  STRUCT
   STAT0 : WORD ;
   STAT1 : WORD ;
   STAT2 : WORD ;
   STAT3 : WORD ;
   STAT4 : WORD ;
   STAT5 : WORD ;
   STAT6 : WORD ;
   STAT7 : WORD ;
   STAT8 : WORD ;
   STAT9 : WORD ;
   STAT10 : WORD ;
   STAT11 : WORD ;
   STAT12 : WORD ;
   STAT13 : WORD ;
   STAT14 : WORD ;
   STAT15 : WORD ;
   STAT16 : INT ;
   STAT17 : INT ;
   STAT18 : INT ;
   STAT19 : INT ;
   STAT20 : ARRAY  [1 .. 6 ] OF BYTE ;
   STAT21 : ARRAY  [1 .. 6 ] OF BYTE ;
   STAT22 : ARRAY  [1 .. 40 ] OF BOOL  := FALSE;
   STAT23 : ARRAY  [1 .. 40 ] OF BOOL  := FALSE;
   STAT24 : WORD ;
   STAT25 : WORD ;
   STAT26 : WORD ;
   STAT27 : WORD ;
   STAT28 : WORD ;
   STAT29 : WORD ;
   STAT30 : WORD ;
   STAT31 : ARRAY  [1 .. 7 ] OF WORD ;
   STAT32 : INT ;
   STAT33 : INT ;
   STAT34 : INT ;
   STAT35 : INT ;
   STAT36 : ARRAY  [1 .. 500 ] OF WORD ;
   STAT37 : ARRAY  [1 .. 16 ] OF BYTE ;
   STAT38 : ARRAY  [1 .. 4 ] OF BYTE ;
   STAT39 : ARRAY  [1 .. 16 ] OF BYTE ;
  END_STRUCT ;
BEGIN
   STAT0 := W#16#2714;
   STAT1 := W#16#87;
   STAT2 := W#16#2222;
   STAT3 := W#16#180;
   STAT4 := W#16#5416;
   STAT5 := W#16#60;
   STAT6 := W#16#0;
   STAT7 := W#16#0;
   STAT8 := W#16#87;
   STAT9 := W#16#2713;
   STAT10 := W#16#220A;
   STAT11 := W#16#8010;
   STAT12 := W#16#5254;
   STAT13 := W#16#4000;
   STAT14 := W#16#0;
   STAT15 := W#16#0;
   STAT16 := 0;
   STAT17 := 2;
   STAT18 := 3;
   STAT19 := 0;
   STAT20[1] := B#16#0;
   STAT20[2] := B#16#0;
   STAT20[3] := B#16#0;
   STAT20[4] := B#16#0;
   STAT20[5] := B#16#0;
   STAT20[6] := B#16#0;
   STAT21[1] := B#16#0;
   STAT21[2] := B#16#0;
   STAT21[3] := B#16#0;
   STAT21[4] := B#16#0;
   STAT21[5] := B#16#0;
   STAT21[6] := B#16#0;
   STAT22[1] := FALSE;
   STAT22[2] := FALSE;
   STAT22[3] := TRUE;
   STAT22[4] := FALSE;
   STAT22[5] := FALSE;
   STAT22[6] := FALSE;
   STAT22[7] := FALSE;
   STAT22[8] := TRUE;
   STAT22[9] := FALSE;
   STAT22[10] := FALSE;
   STAT22[11] := FALSE;
   STAT22[12] := FALSE;
   STAT22[13] := FALSE;
   STAT22[14] := FALSE;
   STAT22[15] := FALSE;
   STAT22[16] := FALSE;
   STAT22[17] := FALSE;
   STAT22[18] := FALSE;
   STAT22[19] := FALSE;
   STAT22[20] := FALSE;
   STAT22[21] := FALSE;
   STAT22[22] := FALSE;
   STAT22[23] := FALSE;
   STAT22[24] := FALSE;
   STAT22[25] := FALSE;
   STAT22[26] := FALSE;
   STAT22[27] := FALSE;
   STAT22[28] := FALSE;
   STAT22[29] := FALSE;
   STAT22[30] := FALSE;
   STAT22[31] := FALSE;
   STAT22[32] := FALSE;
   STAT22[33] := FALSE;
   STAT22[34] := FALSE;
   STAT22[35] := FALSE;
   STAT22[36] := FALSE;
   STAT22[37] := FALSE;
   STAT22[38] := FALSE;
   STAT22[39] := FALSE;
   STAT22[40] := FALSE;
   STAT23[1] := FALSE;
   STAT23[2] := TRUE;
   STAT23[3] := FALSE;
   STAT23[4] := FALSE;
   STAT23[5] := FALSE;
   STAT23[6] := TRUE;
   STAT23[7] := FALSE;
   STAT23[8] := FALSE;
   STAT23[9] := FALSE;
   STAT23[10] := FALSE;
   STAT23[11] := FALSE;
   STAT23[12] := FALSE;
   STAT23[13] := FALSE;
   STAT23[14] := FALSE;
   STAT23[15] := FALSE;
   STAT23[16] := FALSE;
   STAT23[17] := FALSE;
   STAT23[18] := FALSE;
   STAT23[19] := FALSE;
   STAT23[20] := FALSE;
   STAT23[21] := FALSE;
   STAT23[22] := FALSE;
   STAT23[23] := FALSE;
   STAT23[24] := FALSE;
   STAT23[25] := FALSE;
   STAT23[26] := FALSE;
   STAT23[27] := FALSE;
   STAT23[28] := FALSE;
   STAT23[29] := FALSE;
   STAT23[30] := FALSE;
   STAT23[31] := FALSE;
   STAT23[32] := FALSE;
   STAT23[33] := FALSE;
   STAT23[34] := FALSE;
   STAT23[35] := FALSE;
   STAT23[36] := FALSE;
   STAT23[37] := FALSE;
   STAT23[38] := FALSE;
   STAT23[39] := FALSE;
   STAT23[40] := FALSE;
   STAT24 := W#16#400;
   STAT25 := W#16#400;
   STAT26 := W#16#0;
   STAT27 := W#16#0;
   STAT28 := W#16#0;
   STAT29 := W#16#0;
   STAT30 := W#16#0;
   STAT31[1] := W#16#0;
   STAT31[2] := W#16#0;
   STAT31[3] := W#16#0;
   STAT31[4] := W#16#0;
   STAT31[5] := W#16#0;
   STAT31[6] := W#16#0;
   STAT31[7] := W#16#0;
   STAT32 := 100;
   STAT33 := 90;
   STAT34 := 80;
   STAT35 := 0;
   STAT36[1] := W#16#300;
   STAT36[2] := W#16#1418;
   STAT36[3] := W#16#3223;
   STAT36[4] := W#16#B;
   STAT36[5] := W#16#2713;
   STAT36[6] := W#16#200;
   STAT36[7] := W#16#1418;
   STAT36[8] := W#16#3221;
   STAT36[9] := W#16#1;
   STAT36[10] := W#16#2712;
   STAT36[11] := W#16#500;
   STAT36[12] := W#16#1418;
   STAT36[13] := W#16#3221;
   STAT36[14] := W#16#0;
   STAT36[15] := W#16#0;
   STAT36[16] := W#16#400;
   STAT36[17] := W#16#1418;
   STAT36[18] := W#16#3218;
   STAT36[19] := W#16#0;
   STAT36[20] := W#16#0;
   STAT36[21] := W#16#300;
   STAT36[22] := W#16#1418;
   STAT36[23] := W#16#2328;
   STAT36[24] := W#16#B;
   STAT36[25] := W#16#2712;
   STAT36[26] := W#16#200;
   STAT36[27] := W#16#1418;
   STAT36[28] := W#16#2327;
   STAT36[29] := W#16#1;
   STAT36[30] := W#16#2711;
   STAT36[31] := W#16#500;
   STAT36[32] := W#16#1418;
   STAT36[33] := W#16#2327;
   STAT36[34] := W#16#0;
   STAT36[35] := W#16#0;
   STAT36[36] := W#16#400;
   STAT36[37] := W#16#1418;
   STAT36[38] := W#16#2324;
   STAT36[39] := W#16#0;
   STAT36[40] := W#16#0;
   STAT36[41] := W#16#300;
   STAT36[42] := W#16#1418;
   STAT36[43] := W#16#2218;
   STAT36[44] := W#16#B;
   STAT36[45] := W#16#2711;
   STAT36[46] := W#16#200;
   STAT36[47] := W#16#1418;
   STAT36[48] := W#16#2217;
   STAT36[49] := W#16#1;
   STAT36[50] := W#16#2710;
   STAT36[51] := W#16#500;
   STAT36[52] := W#16#1418;
   STAT36[53] := W#16#2217;
   STAT36[54] := W#16#0;
   STAT36[55] := W#16#0;
   STAT36[56] := W#16#400;
   STAT36[57] := W#16#1418;
   STAT36[58] := W#16#2213;
   STAT36[59] := W#16#0;
   STAT36[60] := W#16#0;
   STAT36[61] := W#16#300;
   STAT36[62] := W#16#1418;
   STAT36[63] := W#16#2102;
   STAT36[64] := W#16#B;
   STAT36[65] := W#16#2710;
   STAT36[66] := W#16#200;
   STAT36[67] := W#16#1418;
   STAT36[68] := W#16#2101;
   STAT36[69] := W#16#1;
   STAT36[70] := W#16#2709;
   STAT36[71] := W#16#500;
   STAT36[72] := W#16#1418;
   STAT36[73] := W#16#2101;
   STAT36[74] := W#16#0;
   STAT36[75] := W#16#0;
   STAT36[76] := W#16#400;
   STAT36[77] := W#16#1418;
   STAT36[78] := W#16#2058;
   STAT36[79] := W#16#0;
   STAT36[80] := W#16#0;
   STAT36[81] := W#16#300;
   STAT36[82] := W#16#1418;
   STAT36[83] := W#16#1949;
   STAT36[84] := W#16#B;
   STAT36[85] := W#16#2709;
   STAT36[86] := W#16#200;
   STAT36[87] := W#16#1418;
   STAT36[88] := W#16#1948;
   STAT36[89] := W#16#1;
   STAT36[90] := W#16#2708;
   STAT36[91] := W#16#500;
   STAT36[92] := W#16#1418;
   STAT36[93] := W#16#1947;
   STAT36[94] := W#16#0;
   STAT36[95] := W#16#0;
   STAT36[96] := W#16#400;
   STAT36[97] := W#16#1418;
   STAT36[98] := W#16#1944;
   STAT36[99] := W#16#0;
   STAT36[100] := W#16#0;
   STAT36[101] := W#16#300;
   STAT36[102] := W#16#1418;
   STAT36[103] := W#16#1838;
   STAT36[104] := W#16#B;
   STAT36[105] := W#16#2708;
   STAT36[106] := W#16#200;
   STAT36[107] := W#16#1418;
   STAT36[108] := W#16#1837;
   STAT36[109] := W#16#1;
   STAT36[110] := W#16#2707;
   STAT36[111] := W#16#500;
   STAT36[112] := W#16#1418;
   STAT36[113] := W#16#1836;
   STAT36[114] := W#16#0;
   STAT36[115] := W#16#0;
   STAT36[116] := W#16#400;
   STAT36[117] := W#16#1418;
   STAT36[118] := W#16#1833;
   STAT36[119] := W#16#0;
   STAT36[120] := W#16#0;
   STAT36[121] := W#16#300;
   STAT36[122] := W#16#1418;
   STAT36[123] := W#16#1723;
   STAT36[124] := W#16#B;
   STAT36[125] := W#16#2707;
   STAT36[126] := W#16#200;
   STAT36[127] := W#16#1418;
   STAT36[128] := W#16#1721;
   STAT36[129] := W#16#1;
   STAT36[130] := W#16#2706;
   STAT36[131] := W#16#500;
   STAT36[132] := W#16#1418;
   STAT36[133] := W#16#1721;
   STAT36[134] := W#16#0;
   STAT36[135] := W#16#0;
   STAT36[136] := W#16#400;
   STAT36[137] := W#16#1418;
   STAT36[138] := W#16#1718;
   STAT36[139] := W#16#0;
   STAT36[140] := W#16#0;
   STAT36[141] := W#16#300;
   STAT36[142] := W#16#1418;
   STAT36[143] := W#16#1610;
   STAT36[144] := W#16#B;
   STAT36[145] := W#16#2706;
   STAT36[146] := W#16#200;
   STAT36[147] := W#16#1418;
   STAT36[148] := W#16#1609;
   STAT36[149] := W#16#1;
   STAT36[150] := W#16#2705;
   STAT36[151] := W#16#500;
   STAT36[152] := W#16#1418;
   STAT36[153] := W#16#1608;
   STAT36[154] := W#16#0;
   STAT36[155] := W#16#0;
   STAT36[156] := W#16#400;
   STAT36[157] := W#16#1418;
   STAT36[158] := W#16#1605;
   STAT36[159] := W#16#0;
   STAT36[160] := W#16#0;
   STAT36[161] := W#16#300;
   STAT36[162] := W#16#1418;
   STAT36[163] := W#16#1459;
   STAT36[164] := W#16#B;
   STAT36[165] := W#16#2705;
   STAT36[166] := W#16#200;
   STAT36[167] := W#16#1418;
   STAT36[168] := W#16#1458;
   STAT36[169] := W#16#1;
   STAT36[170] := W#16#2704;
   STAT36[171] := W#16#500;
   STAT36[172] := W#16#1418;
   STAT36[173] := W#16#1457;
   STAT36[174] := W#16#0;
   STAT36[175] := W#16#0;
   STAT36[176] := W#16#400;
   STAT36[177] := W#16#1418;
   STAT36[178] := W#16#1454;
   STAT36[179] := W#16#0;
   STAT36[180] := W#16#0;
   STAT36[181] := W#16#300;
   STAT36[182] := W#16#1418;
   STAT36[183] := W#16#1343;
   STAT36[184] := W#16#B;
   STAT36[185] := W#16#2704;
   STAT36[186] := W#16#200;
   STAT36[187] := W#16#1418;
   STAT36[188] := W#16#1342;
   STAT36[189] := W#16#1;
   STAT36[190] := W#16#2703;
   STAT36[191] := W#16#500;
   STAT36[192] := W#16#1418;
   STAT36[193] := W#16#1342;
   STAT36[194] := W#16#0;
   STAT36[195] := W#16#0;
   STAT36[196] := W#16#400;
   STAT36[197] := W#16#1418;
   STAT36[198] := W#16#1338;
   STAT36[199] := W#16#0;
   STAT36[200] := W#16#0;
   STAT36[201] := W#16#300;
   STAT36[202] := W#16#1418;
   STAT36[203] := W#16#1228;
   STAT36[204] := W#16#B;
   STAT36[205] := W#16#2703;
   STAT36[206] := W#16#200;
   STAT36[207] := W#16#1418;
   STAT36[208] := W#16#1226;
   STAT36[209] := W#16#1;
   STAT36[210] := W#16#2702;
   STAT36[211] := W#16#500;
   STAT36[212] := W#16#1418;
   STAT36[213] := W#16#1226;
   STAT36[214] := W#16#0;
   STAT36[215] := W#16#0;
   STAT36[216] := W#16#400;
   STAT36[217] := W#16#1418;
   STAT36[218] := W#16#1223;
   STAT36[219] := W#16#0;
   STAT36[220] := W#16#0;
   STAT36[221] := W#16#300;
   STAT36[222] := W#16#1418;
   STAT36[223] := W#16#1112;
   STAT36[224] := W#16#B;
   STAT36[225] := W#16#2702;
   STAT36[226] := W#16#200;
   STAT36[227] := W#16#1418;
   STAT36[228] := W#16#1111;
   STAT36[229] := W#16#1;
   STAT36[230] := W#16#2701;
   STAT36[231] := W#16#500;
   STAT36[232] := W#16#1418;
   STAT36[233] := W#16#1110;
   STAT36[234] := W#16#0;
   STAT36[235] := W#16#0;
   STAT36[236] := W#16#400;
   STAT36[237] := W#16#1418;
   STAT36[238] := W#16#1107;
   STAT36[239] := W#16#0;
   STAT36[240] := W#16#0;
   STAT36[241] := W#16#300;
   STAT36[242] := W#16#1418;
   STAT36[243] := W#16#957;
   STAT36[244] := W#16#B;
   STAT36[245] := W#16#2701;
   STAT36[246] := W#16#200;
   STAT36[247] := W#16#1418;
   STAT36[248] := W#16#955;
   STAT36[249] := W#16#1;
   STAT36[250] := W#16#2700;
   STAT36[251] := W#16#500;
   STAT36[252] := W#16#1418;
   STAT36[253] := W#16#955;
   STAT36[254] := W#16#0;
   STAT36[255] := W#16#0;
   STAT36[256] := W#16#400;
   STAT36[257] := W#16#1418;
   STAT36[258] := W#16#952;
   STAT36[259] := W#16#0;
   STAT36[260] := W#16#0;
   STAT36[261] := W#16#300;
   STAT36[262] := W#16#1418;
   STAT36[263] := W#16#844;
   STAT36[264] := W#16#B;
   STAT36[265] := W#16#2700;
   STAT36[266] := W#16#200;
   STAT36[267] := W#16#1418;
   STAT36[268] := W#16#843;
   STAT36[269] := W#16#1;
   STAT36[270] := W#16#2699;
   STAT36[271] := W#16#500;
   STAT36[272] := W#16#1418;
   STAT36[273] := W#16#842;
   STAT36[274] := W#16#0;
   STAT36[275] := W#16#0;
   STAT36[276] := W#16#400;
   STAT36[277] := W#16#1418;
   STAT36[278] := W#16#839;
   STAT36[279] := W#16#0;
   STAT36[280] := W#16#0;
   STAT36[281] := W#16#300;
   STAT36[282] := W#16#1418;
   STAT36[283] := W#16#729;
   STAT36[284] := W#16#B;
   STAT36[285] := W#16#2699;
   STAT36[286] := W#16#200;
   STAT36[287] := W#16#1418;
   STAT36[288] := W#16#728;
   STAT36[289] := W#16#1;
   STAT36[290] := W#16#2698;
   STAT36[291] := W#16#500;
   STAT36[292] := W#16#1418;
   STAT36[293] := W#16#728;
   STAT36[294] := W#16#0;
   STAT36[295] := W#16#0;
   STAT36[296] := W#16#400;
   STAT36[297] := W#16#1418;
   STAT36[298] := W#16#724;
   STAT36[299] := W#16#0;
   STAT36[300] := W#16#0;
   STAT36[301] := W#16#300;
   STAT36[302] := W#16#1418;
   STAT36[303] := W#16#324;
   STAT36[304] := W#16#B;
   STAT36[305] := W#16#2698;
   STAT36[306] := W#16#200;
   STAT36[307] := W#16#1418;
   STAT36[308] := W#16#322;
   STAT36[309] := W#16#1;
   STAT36[310] := W#16#2697;
   STAT36[311] := W#16#500;
   STAT36[312] := W#16#1418;
   STAT36[313] := W#16#322;
   STAT36[314] := W#16#0;
   STAT36[315] := W#16#0;
   STAT36[316] := W#16#400;
   STAT36[317] := W#16#1418;
   STAT36[318] := W#16#319;
   STAT36[319] := W#16#0;
   STAT36[320] := W#16#0;
   STAT36[321] := W#16#300;
   STAT36[322] := W#16#1418;
   STAT36[323] := W#16#211;
   STAT36[324] := W#16#B;
   STAT36[325] := W#16#2697;
   STAT36[326] := W#16#200;
   STAT36[327] := W#16#1418;
   STAT36[328] := W#16#209;
   STAT36[329] := W#16#1;
   STAT36[330] := W#16#2696;
   STAT36[331] := W#16#500;
   STAT36[332] := W#16#1418;
   STAT36[333] := W#16#209;
   STAT36[334] := W#16#0;
   STAT36[335] := W#16#0;
   STAT36[336] := W#16#400;
   STAT36[337] := W#16#1418;
   STAT36[338] := W#16#206;
   STAT36[339] := W#16#0;
   STAT36[340] := W#16#0;
   STAT36[341] := W#16#300;
   STAT36[342] := W#16#1418;
   STAT36[343] := W#16#55;
   STAT36[344] := W#16#B;
   STAT36[345] := W#16#2696;
   STAT36[346] := W#16#200;
   STAT36[347] := W#16#1418;
   STAT36[348] := W#16#53;
   STAT36[349] := W#16#1;
   STAT36[350] := W#16#2695;
   STAT36[351] := W#16#500;
   STAT36[352] := W#16#1418;
   STAT36[353] := W#16#53;
   STAT36[354] := W#16#0;
   STAT36[355] := W#16#0;
   STAT36[356] := W#16#400;
   STAT36[357] := W#16#1418;
   STAT36[358] := W#16#50;
   STAT36[359] := W#16#0;
   STAT36[360] := W#16#0;
   STAT36[361] := W#16#300;
   STAT36[362] := W#16#1417;
   STAT36[363] := W#16#5939;
   STAT36[364] := W#16#B;
   STAT36[365] := W#16#2695;
   STAT36[366] := W#16#200;
   STAT36[367] := W#16#1417;
   STAT36[368] := W#16#5938;
   STAT36[369] := W#16#1;
   STAT36[370] := W#16#2694;
   STAT36[371] := W#16#500;
   STAT36[372] := W#16#1417;
   STAT36[373] := W#16#5937;
   STAT36[374] := W#16#0;
   STAT36[375] := W#16#0;
   STAT36[376] := W#16#400;
   STAT36[377] := W#16#1417;
   STAT36[378] := W#16#5934;
   STAT36[379] := W#16#0;
   STAT36[380] := W#16#0;
   STAT36[381] := W#16#300;
   STAT36[382] := W#16#1417;
   STAT36[383] := W#16#5828;
   STAT36[384] := W#16#B;
   STAT36[385] := W#16#2694;
   STAT36[386] := W#16#200;
   STAT36[387] := W#16#1417;
   STAT36[388] := W#16#5827;
   STAT36[389] := W#16#1;
   STAT36[390] := W#16#2693;
   STAT36[391] := W#16#500;
   STAT36[392] := W#16#1417;
   STAT36[393] := W#16#5827;
   STAT36[394] := W#16#0;
   STAT36[395] := W#16#0;
   STAT36[396] := W#16#400;
   STAT36[397] := W#16#1417;
   STAT36[398] := W#16#5824;
   STAT36[399] := W#16#0;
   STAT36[400] := W#16#0;
   STAT36[401] := W#16#300;
   STAT36[402] := W#16#1417;
   STAT36[403] := W#16#5715;
   STAT36[404] := W#16#B;
   STAT36[405] := W#16#2693;
   STAT36[406] := W#16#200;
   STAT36[407] := W#16#1417;
   STAT36[408] := W#16#5714;
   STAT36[409] := W#16#1;
   STAT36[410] := W#16#2692;
   STAT36[411] := W#16#500;
   STAT36[412] := W#16#1417;
   STAT36[413] := W#16#5713;
   STAT36[414] := W#16#0;
   STAT36[415] := W#16#0;
   STAT36[416] := W#16#400;
   STAT36[417] := W#16#1417;
   STAT36[418] := W#16#5710;
   STAT36[419] := W#16#0;
   STAT36[420] := W#16#0;
   STAT36[421] := W#16#300;
   STAT36[422] := W#16#1417;
   STAT36[423] := W#16#5602;
   STAT36[424] := W#16#B;
   STAT36[425] := W#16#2692;
   STAT36[426] := W#16#200;
   STAT36[427] := W#16#1417;
   STAT36[428] := W#16#5601;
   STAT36[429] := W#16#1;
   STAT36[430] := W#16#2691;
   STAT36[431] := W#16#500;
   STAT36[432] := W#16#1417;
   STAT36[433] := W#16#5600;
   STAT36[434] := W#16#0;
   STAT36[435] := W#16#0;
   STAT36[436] := W#16#400;
   STAT36[437] := W#16#1417;
   STAT36[438] := W#16#5557;
   STAT36[439] := W#16#0;
   STAT36[440] := W#16#0;
   STAT36[441] := W#16#300;
   STAT36[442] := W#16#1417;
   STAT36[443] := W#16#5448;
   STAT36[444] := W#16#B;
   STAT36[445] := W#16#2691;
   STAT36[446] := W#16#200;
   STAT36[447] := W#16#1417;
   STAT36[448] := W#16#5447;
   STAT36[449] := W#16#1;
   STAT36[450] := W#16#2690;
   STAT36[451] := W#16#500;
   STAT36[452] := W#16#1417;
   STAT36[453] := W#16#5447;
   STAT36[454] := W#16#0;
   STAT36[455] := W#16#0;
   STAT36[456] := W#16#400;
   STAT36[457] := W#16#1417;
   STAT36[458] := W#16#5444;
   STAT36[459] := W#16#0;
   STAT36[460] := W#16#0;
   STAT36[461] := W#16#300;
   STAT36[462] := W#16#1417;
   STAT36[463] := W#16#5333;
   STAT36[464] := W#16#B;
   STAT36[465] := W#16#2690;
   STAT36[466] := W#16#200;
   STAT36[467] := W#16#1417;
   STAT36[468] := W#16#5331;
   STAT36[469] := W#16#1;
   STAT36[470] := W#16#2689;
   STAT36[471] := W#16#500;
   STAT36[472] := W#16#1417;
   STAT36[473] := W#16#5331;
   STAT36[474] := W#16#0;
   STAT36[475] := W#16#0;
   STAT36[476] := W#16#400;
   STAT36[477] := W#16#1417;
   STAT36[478] := W#16#5328;
   STAT36[479] := W#16#0;
   STAT36[480] := W#16#0;
   STAT36[481] := W#16#300;
   STAT36[482] := W#16#1417;
   STAT36[483] := W#16#5217;
   STAT36[484] := W#16#B;
   STAT36[485] := W#16#2689;
   STAT36[486] := W#16#200;
   STAT36[487] := W#16#1417;
   STAT36[488] := W#16#5216;
   STAT36[489] := W#16#1;
   STAT36[490] := W#16#2688;
   STAT36[491] := W#16#500;
   STAT36[492] := W#16#1417;
   STAT36[493] := W#16#5215;
   STAT36[494] := W#16#0;
   STAT36[495] := W#16#0;
   STAT36[496] := W#16#400;
   STAT36[497] := W#16#1417;
   STAT36[498] := W#16#5212;
   STAT36[499] := W#16#0;
   STAT36[500] := W#16#0;
   STAT37[1] := B#16#0;
   STAT37[2] := B#16#87;
   STAT37[3] := B#16#27;
   STAT37[4] := B#16#13;
   STAT37[5] := B#16#22;
   STAT37[6] := B#16#A;
   STAT37[7] := B#16#80;
   STAT37[8] := B#16#10;
   STAT37[9] := B#16#52;
   STAT37[10] := B#16#54;
   STAT37[11] := B#16#40;
   STAT37[12] := B#16#0;
   STAT37[13] := B#16#0;
   STAT37[14] := B#16#0;
   STAT37[15] := B#16#0;
   STAT37[16] := B#16#0;
   STAT38[1] := B#16#0;
   STAT38[2] := B#16#0;
   STAT38[3] := B#16#0;
   STAT38[4] := B#16#0;
   STAT39[1] := B#16#27;
   STAT39[2] := B#16#13;
   STAT39[3] := B#16#0;
   STAT39[4] := B#16#87;
   STAT39[5] := B#16#A;
   STAT39[6] := B#16#22;
   STAT39[7] := B#16#10;
   STAT39[8] := B#16#80;
   STAT39[9] := B#16#54;
   STAT39[10] := B#16#52;
   STAT39[11] := B#16#0;
   STAT39[12] := B#16#40;
   STAT39[13] := B#16#0;
   STAT39[14] := B#16#0;
   STAT39[15] := B#16#0;
   STAT39[16] := B#16#0;
END_DATA_BLOCK

DATA_BLOCK DB 169
VERSION : 0.1


  STRUCT
   STAT0 : WORD ;
   STAT1 : WORD ;
   STAT2 : WORD ;
   STAT3 : WORD ;
   STAT4 : WORD ;
   STAT5 : WORD ;
   STAT6 : WORD ;
   STAT7 : WORD ;
   STAT8 : WORD ;
   STAT9 : WORD ;
   STAT10 : WORD ;
   STAT11 : WORD ;
   STAT12 : WORD ;
   STAT13 : WORD ;
   STAT14 : WORD ;
   STAT15 : WORD ;
   STAT16 : INT ;
   STAT17 : INT ;
   STAT18 : INT ;
   STAT19 : INT ;
   STAT20 : ARRAY  [1 .. 6 ] OF BYTE ;
   STAT21 : ARRAY  [1 .. 6 ] OF BYTE ;
   STAT22 : ARRAY  [1 .. 40 ] OF BOOL  := FALSE;
   STAT23 : ARRAY  [1 .. 40 ] OF BOOL  := FALSE;
   STAT24 : WORD ;
   STAT25 : WORD ;
   STAT26 : WORD ;
   STAT27 : WORD ;
   STAT28 : WORD ;
   STAT29 : WORD ;
   STAT30 : WORD ;
   STAT31 : ARRAY  [1 .. 7 ] OF WORD ;
   STAT32 : INT ;
   STAT33 : INT ;
   STAT34 : INT ;
   STAT35 : INT ;
   STAT36 : ARRAY  [1 .. 500 ] OF WORD ;
   STAT37 : ARRAY  [1 .. 16 ] OF BYTE ;
   STAT38 : ARRAY  [1 .. 4 ] OF BYTE ;
   STAT39 : ARRAY  [1 .. 16 ] OF BYTE ;
  END_STRUCT ;
BEGIN
   STAT0 := W#16#2705;
   STAT1 := W#16#87;
   STAT2 := W#16#A22;
   STAT3 := W#16#1080;
   STAT4 := W#16#1026;
   STAT5 := W#16#40;
   STAT6 := W#16#0;
   STAT7 := W#16#0;
   STAT8 := W#16#87;
   STAT9 := W#16#2709;
   STAT10 := W#16#220A;
   STAT11 := W#16#8010;
   STAT12 := W#16#1610;
   STAT13 := W#16#4000;
   STAT14 := W#16#0;
   STAT15 := W#16#0;
   STAT16 := 2;
   STAT17 := 8;
   STAT18 := 3;
   STAT19 := 0;
   STAT20[1] := B#16#0;
   STAT20[2] := B#16#0;
   STAT20[3] := B#16#0;
   STAT20[4] := B#16#0;
   STAT20[5] := B#16#0;
   STAT20[6] := B#16#0;
   STAT21[1] := B#16#0;
   STAT21[2] := B#16#0;
   STAT21[3] := B#16#0;
   STAT21[4] := B#16#0;
   STAT21[5] := B#16#0;
   STAT21[6] := B#16#0;
   STAT22[1] := FALSE;
   STAT22[2] := FALSE;
   STAT22[3] := TRUE;
   STAT22[4] := FALSE;
   STAT22[5] := FALSE;
   STAT22[6] := FALSE;
   STAT22[7] := FALSE;
   STAT22[8] := TRUE;
   STAT22[9] := FALSE;
   STAT22[10] := FALSE;
   STAT22[11] := FALSE;
   STAT22[12] := FALSE;
   STAT22[13] := FALSE;
   STAT22[14] := FALSE;
   STAT22[15] := FALSE;
   STAT22[16] := FALSE;
   STAT22[17] := FALSE;
   STAT22[18] := FALSE;
   STAT22[19] := FALSE;
   STAT22[20] := FALSE;
   STAT22[21] := FALSE;
   STAT22[22] := FALSE;
   STAT22[23] := FALSE;
   STAT22[24] := FALSE;
   STAT22[25] := FALSE;
   STAT22[26] := FALSE;
   STAT22[27] := FALSE;
   STAT22[28] := FALSE;
   STAT22[29] := FALSE;
   STAT22[30] := FALSE;
   STAT22[31] := FALSE;
   STAT22[32] := FALSE;
   STAT22[33] := FALSE;
   STAT22[34] := FALSE;
   STAT22[35] := FALSE;
   STAT22[36] := FALSE;
   STAT22[37] := FALSE;
   STAT22[38] := FALSE;
   STAT22[39] := FALSE;
   STAT22[40] := FALSE;
   STAT23[1] := TRUE;
   STAT23[2] := FALSE;
   STAT23[3] := TRUE;
   STAT23[4] := TRUE;
   STAT23[5] := TRUE;
   STAT23[6] := FALSE;
   STAT23[7] := FALSE;
   STAT23[8] := FALSE;
   STAT23[9] := FALSE;
   STAT23[10] := FALSE;
   STAT23[11] := FALSE;
   STAT23[12] := FALSE;
   STAT23[13] := FALSE;
   STAT23[14] := FALSE;
   STAT23[15] := FALSE;
   STAT23[16] := FALSE;
   STAT23[17] := FALSE;
   STAT23[18] := FALSE;
   STAT23[19] := FALSE;
   STAT23[20] := FALSE;
   STAT23[21] := FALSE;
   STAT23[22] := FALSE;
   STAT23[23] := FALSE;
   STAT23[24] := FALSE;
   STAT23[25] := FALSE;
   STAT23[26] := TRUE;
   STAT23[27] := FALSE;
   STAT23[28] := FALSE;
   STAT23[29] := FALSE;
   STAT23[30] := FALSE;
   STAT23[31] := FALSE;
   STAT23[32] := FALSE;
   STAT23[33] := FALSE;
   STAT23[34] := FALSE;
   STAT23[35] := FALSE;
   STAT23[36] := FALSE;
   STAT23[37] := FALSE;
   STAT23[38] := FALSE;
   STAT23[39] := FALSE;
   STAT23[40] := FALSE;
   STAT24 := W#16#0;
   STAT25 := W#16#0;
   STAT26 := W#16#0;
   STAT27 := W#16#0;
   STAT28 := W#16#0;
   STAT29 := W#16#0;
   STAT30 := W#16#0;
   STAT31[1] := W#16#0;
   STAT31[2] := W#16#0;
   STAT31[3] := W#16#0;
   STAT31[4] := W#16#0;
   STAT31[5] := W#16#0;
   STAT31[6] := W#16#0;
   STAT31[7] := W#16#0;
   STAT32 := 100;
   STAT33 := 90;
   STAT34 := 80;
   STAT35 := 0;
   STAT36[1] := W#16#400;
   STAT36[2] := W#16#1418;
   STAT36[3] := W#16#3243;
   STAT36[4] := W#16#0;
   STAT36[5] := W#16#2709;
   STAT36[6] := W#16#300;
   STAT36[7] := W#16#1418;
   STAT36[8] := W#16#3240;
   STAT36[9] := W#16#B;
   STAT36[10] := W#16#2705;
   STAT36[11] := W#16#200;
   STAT36[12] := W#16#1418;
   STAT36[13] := W#16#3238;
   STAT36[14] := W#16#1;
   STAT36[15] := W#16#0;
   STAT36[16] := W#16#500;
   STAT36[17] := W#16#1418;
   STAT36[18] := W#16#3229;
   STAT36[19] := W#16#0;
   STAT36[20] := W#16#0;
   STAT36[21] := W#16#400;
   STAT36[22] := W#16#1418;
   STAT36[23] := W#16#3229;
   STAT36[24] := W#16#0;
   STAT36[25] := W#16#0;
   STAT36[26] := W#16#500;
   STAT36[27] := W#16#1418;
   STAT36[28] := W#16#3228;
   STAT36[29] := W#16#0;
   STAT36[30] := W#16#0;
   STAT36[31] := W#16#400;
   STAT36[32] := W#16#1418;
   STAT36[33] := W#16#3128;
   STAT36[34] := W#16#0;
   STAT36[35] := W#16#2708;
   STAT36[36] := W#16#300;
   STAT36[37] := W#16#1418;
   STAT36[38] := W#16#3125;
   STAT36[39] := W#16#B;
   STAT36[40] := W#16#2704;
   STAT36[41] := W#16#200;
   STAT36[42] := W#16#1418;
   STAT36[43] := W#16#3124;
   STAT36[44] := W#16#1;
   STAT36[45] := W#16#0;
   STAT36[46] := W#16#500;
   STAT36[47] := W#16#1418;
   STAT36[48] := W#16#3115;
   STAT36[49] := W#16#0;
   STAT36[50] := W#16#0;
   STAT36[51] := W#16#400;
   STAT36[52] := W#16#1418;
   STAT36[53] := W#16#3114;
   STAT36[54] := W#16#0;
   STAT36[55] := W#16#0;
   STAT36[56] := W#16#500;
   STAT36[57] := W#16#1418;
   STAT36[58] := W#16#3113;
   STAT36[59] := W#16#0;
   STAT36[60] := W#16#0;
   STAT36[61] := W#16#400;
   STAT36[62] := W#16#1418;
   STAT36[63] := W#16#2233;
   STAT36[64] := W#16#0;
   STAT36[65] := W#16#2707;
   STAT36[66] := W#16#300;
   STAT36[67] := W#16#1418;
   STAT36[68] := W#16#2231;
   STAT36[69] := W#16#B;
   STAT36[70] := W#16#2703;
   STAT36[71] := W#16#200;
   STAT36[72] := W#16#1418;
   STAT36[73] := W#16#2229;
   STAT36[74] := W#16#1;
   STAT36[75] := W#16#0;
   STAT36[76] := W#16#500;
   STAT36[77] := W#16#1418;
   STAT36[78] := W#16#2217;
   STAT36[79] := W#16#0;
   STAT36[80] := W#16#0;
   STAT36[81] := W#16#400;
   STAT36[82] := W#16#1418;
   STAT36[83] := W#16#2216;
   STAT36[84] := W#16#0;
   STAT36[85] := W#16#0;
   STAT36[86] := W#16#500;
   STAT36[87] := W#16#1418;
   STAT36[88] := W#16#2215;
   STAT36[89] := W#16#0;
   STAT36[90] := W#16#0;
   STAT36[91] := W#16#400;
   STAT36[92] := W#16#1418;
   STAT36[93] := W#16#2123;
   STAT36[94] := W#16#0;
   STAT36[95] := W#16#2706;
   STAT36[96] := W#16#300;
   STAT36[97] := W#16#1418;
   STAT36[98] := W#16#2120;
   STAT36[99] := W#16#B;
   STAT36[100] := W#16#2702;
   STAT36[101] := W#16#200;
   STAT36[102] := W#16#1418;
   STAT36[103] := W#16#2119;
   STAT36[104] := W#16#1;
   STAT36[105] := W#16#0;
   STAT36[106] := W#16#500;
   STAT36[107] := W#16#1418;
   STAT36[108] := W#16#2103;
   STAT36[109] := W#16#0;
   STAT36[110] := W#16#0;
   STAT36[111] := W#16#400;
   STAT36[112] := W#16#1418;
   STAT36[113] := W#16#2007;
   STAT36[114] := W#16#0;
   STAT36[115] := W#16#2705;
   STAT36[116] := W#16#300;
   STAT36[117] := W#16#1418;
   STAT36[118] := W#16#2004;
   STAT36[119] := W#16#B;
   STAT36[120] := W#16#2701;
   STAT36[121] := W#16#200;
   STAT36[122] := W#16#1418;
   STAT36[123] := W#16#2003;
   STAT36[124] := W#16#1;
   STAT36[125] := W#16#0;
   STAT36[126] := W#16#500;
   STAT36[127] := W#16#1418;
   STAT36[128] := W#16#1949;
   STAT36[129] := W#16#0;
   STAT36[130] := W#16#0;
   STAT36[131] := W#16#400;
   STAT36[132] := W#16#1418;
   STAT36[133] := W#16#1948;
   STAT36[134] := W#16#0;
   STAT36[135] := W#16#0;
   STAT36[136] := W#16#500;
   STAT36[137] := W#16#1418;
   STAT36[138] := W#16#1947;
   STAT36[139] := W#16#0;
   STAT36[140] := W#16#0;
   STAT36[141] := W#16#400;
   STAT36[142] := W#16#1418;
   STAT36[143] := W#16#1854;
   STAT36[144] := W#16#0;
   STAT36[145] := W#16#2704;
   STAT36[146] := W#16#300;
   STAT36[147] := W#16#1418;
   STAT36[148] := W#16#1851;
   STAT36[149] := W#16#B;
   STAT36[150] := W#16#2700;
   STAT36[151] := W#16#200;
   STAT36[152] := W#16#1418;
   STAT36[153] := W#16#1849;
   STAT36[154] := W#16#1;
   STAT36[155] := W#16#0;
   STAT36[156] := W#16#500;
   STAT36[157] := W#16#1418;
   STAT36[158] := W#16#1833;
   STAT36[159] := W#16#0;
   STAT36[160] := W#16#0;
   STAT36[161] := W#16#400;
   STAT36[162] := W#16#1418;
   STAT36[163] := W#16#1833;
   STAT36[164] := W#16#0;
   STAT36[165] := W#16#0;
   STAT36[166] := W#16#500;
   STAT36[167] := W#16#1418;
   STAT36[168] := W#16#1832;
   STAT36[169] := W#16#0;
   STAT36[170] := W#16#0;
   STAT36[171] := W#16#400;
   STAT36[172] := W#16#1418;
   STAT36[173] := W#16#1743;
   STAT36[174] := W#16#0;
   STAT36[175] := W#16#2703;
   STAT36[176] := W#16#300;
   STAT36[177] := W#16#1418;
   STAT36[178] := W#16#1740;
   STAT36[179] := W#16#B;
   STAT36[180] := W#16#2699;
   STAT36[181] := W#16#200;
   STAT36[182] := W#16#1418;
   STAT36[183] := W#16#1739;
   STAT36[184] := W#16#1;
   STAT36[185] := W#16#0;
   STAT36[186] := W#16#500;
   STAT36[187] := W#16#1418;
   STAT36[188] := W#16#1721;
   STAT36[189] := W#16#0;
   STAT36[190] := W#16#0;
   STAT36[191] := W#16#400;
   STAT36[192] := W#16#1418;
   STAT36[193] := W#16#1720;
   STAT36[194] := W#16#0;
   STAT36[195] := W#16#0;
   STAT36[196] := W#16#500;
   STAT36[197] := W#16#1418;
   STAT36[198] := W#16#1719;
   STAT36[199] := W#16#0;
   STAT36[200] := W#16#0;
   STAT36[201] := W#16#400;
   STAT36[202] := W#16#1418;
   STAT36[203] := W#16#1627;
   STAT36[204] := W#16#0;
   STAT36[205] := W#16#2702;
   STAT36[206] := W#16#300;
   STAT36[207] := W#16#1418;
   STAT36[208] := W#16#1625;
   STAT36[209] := W#16#B;
   STAT36[210] := W#16#2698;
   STAT36[211] := W#16#200;
   STAT36[212] := W#16#1418;
   STAT36[213] := W#16#1623;
   STAT36[214] := W#16#1;
   STAT36[215] := W#16#0;
   STAT36[216] := W#16#500;
   STAT36[217] := W#16#1418;
   STAT36[218] := W#16#1607;
   STAT36[219] := W#16#0;
   STAT36[220] := W#16#0;
   STAT36[221] := W#16#400;
   STAT36[222] := W#16#1418;
   STAT36[223] := W#16#1607;
   STAT36[224] := W#16#0;
   STAT36[225] := W#16#0;
   STAT36[226] := W#16#500;
   STAT36[227] := W#16#1418;
   STAT36[228] := W#16#1606;
   STAT36[229] := W#16#0;
   STAT36[230] := W#16#0;
   STAT36[231] := W#16#400;
   STAT36[232] := W#16#1418;
   STAT36[233] := W#16#1514;
   STAT36[234] := W#16#0;
   STAT36[235] := W#16#2701;
   STAT36[236] := W#16#300;
   STAT36[237] := W#16#1418;
   STAT36[238] := W#16#1511;
   STAT36[239] := W#16#B;
   STAT36[240] := W#16#2697;
   STAT36[241] := W#16#200;
   STAT36[242] := W#16#1418;
   STAT36[243] := W#16#1510;
   STAT36[244] := W#16#1;
   STAT36[245] := W#16#0;
   STAT36[246] := W#16#500;
   STAT36[247] := W#16#1418;
   STAT36[248] := W#16#1454;
   STAT36[249] := W#16#0;
   STAT36[250] := W#16#0;
   STAT36[251] := W#16#400;
   STAT36[252] := W#16#1418;
   STAT36[253] := W#16#1454;
   STAT36[254] := W#16#0;
   STAT36[255] := W#16#0;
   STAT36[256] := W#16#500;
   STAT36[257] := W#16#1418;
   STAT36[258] := W#16#1453;
   STAT36[259] := W#16#0;
   STAT36[260] := W#16#0;
   STAT36[261] := W#16#400;
   STAT36[262] := W#16#1418;
   STAT36[263] := W#16#1404;
   STAT36[264] := W#16#0;
   STAT36[265] := W#16#2700;
   STAT36[266] := W#16#300;
   STAT36[267] := W#16#1418;
   STAT36[268] := W#16#1401;
   STAT36[269] := W#16#B;
   STAT36[270] := W#16#2696;
   STAT36[271] := W#16#200;
   STAT36[272] := W#16#1418;
   STAT36[273] := W#16#1359;
   STAT36[274] := W#16#1;
   STAT36[275] := W#16#0;
   STAT36[276] := W#16#500;
   STAT36[277] := W#16#1418;
   STAT36[278] := W#16#1342;
   STAT36[279] := W#16#0;
   STAT36[280] := W#16#0;
   STAT36[281] := W#16#400;
   STAT36[282] := W#16#1418;
   STAT36[283] := W#16#1342;
   STAT36[284] := W#16#0;
   STAT36[285] := W#16#0;
   STAT36[286] := W#16#500;
   STAT36[287] := W#16#1418;
   STAT36[288] := W#16#1340;
   STAT36[289] := W#16#0;
   STAT36[290] := W#16#0;
   STAT36[291] := W#16#400;
   STAT36[292] := W#16#1418;
   STAT36[293] := W#16#1248;
   STAT36[294] := W#16#0;
   STAT36[295] := W#16#2699;
   STAT36[296] := W#16#300;
   STAT36[297] := W#16#1418;
   STAT36[298] := W#16#1245;
   STAT36[299] := W#16#B;
   STAT36[300] := W#16#2695;
   STAT36[301] := W#16#200;
   STAT36[302] := W#16#1418;
   STAT36[303] := W#16#1244;
   STAT36[304] := W#16#1;
   STAT36[305] := W#16#0;
   STAT36[306] := W#16#500;
   STAT36[307] := W#16#1418;
   STAT36[308] := W#16#1228;
   STAT36[309] := W#16#0;
   STAT36[310] := W#16#0;
   STAT36[311] := W#16#400;
   STAT36[312] := W#16#1418;
   STAT36[313] := W#16#1227;
   STAT36[314] := W#16#0;
   STAT36[315] := W#16#0;
   STAT36[316] := W#16#500;
   STAT36[317] := W#16#1418;
   STAT36[318] := W#16#1226;
   STAT36[319] := W#16#0;
   STAT36[320] := W#16#0;
   STAT36[321] := W#16#400;
   STAT36[322] := W#16#1418;
   STAT36[323] := W#16#1132;
   STAT36[324] := W#16#0;
   STAT36[325] := W#16#2698;
   STAT36[326] := W#16#300;
   STAT36[327] := W#16#1418;
   STAT36[328] := W#16#1130;
   STAT36[329] := W#16#B;
   STAT36[330] := W#16#2694;
   STAT36[331] := W#16#200;
   STAT36[332] := W#16#1418;
   STAT36[333] := W#16#1128;
   STAT36[334] := W#16#1;
   STAT36[335] := W#16#0;
   STAT36[336] := W#16#500;
   STAT36[337] := W#16#1418;
   STAT36[338] := W#16#1115;
   STAT36[339] := W#16#0;
   STAT36[340] := W#16#0;
   STAT36[341] := W#16#400;
   STAT36[342] := W#16#1418;
   STAT36[343] := W#16#1114;
   STAT36[344] := W#16#0;
   STAT36[345] := W#16#0;
   STAT36[346] := W#16#500;
   STAT36[347] := W#16#1418;
   STAT36[348] := W#16#1113;
   STAT36[349] := W#16#0;
   STAT36[350] := W#16#0;
   STAT36[351] := W#16#400;
   STAT36[352] := W#16#1418;
   STAT36[353] := W#16#1016;
   STAT36[354] := W#16#0;
   STAT36[355] := W#16#2697;
   STAT36[356] := W#16#300;
   STAT36[357] := W#16#1418;
   STAT36[358] := W#16#1014;
   STAT36[359] := W#16#B;
   STAT36[360] := W#16#2693;
   STAT36[361] := W#16#200;
   STAT36[362] := W#16#1418;
   STAT36[363] := W#16#1012;
   STAT36[364] := W#16#1;
   STAT36[365] := W#16#0;
   STAT36[366] := W#16#500;
   STAT36[367] := W#16#1418;
   STAT36[368] := W#16#1002;
   STAT36[369] := W#16#0;
   STAT36[370] := W#16#0;
   STAT36[371] := W#16#400;
   STAT36[372] := W#16#1418;
   STAT36[373] := W#16#901;
   STAT36[374] := W#16#0;
   STAT36[375] := W#16#2696;
   STAT36[376] := W#16#300;
   STAT36[377] := W#16#1418;
   STAT36[378] := W#16#858;
   STAT36[379] := W#16#B;
   STAT36[380] := W#16#2692;
   STAT36[381] := W#16#200;
   STAT36[382] := W#16#1418;
   STAT36[383] := W#16#857;
   STAT36[384] := W#16#1;
   STAT36[385] := W#16#0;
   STAT36[386] := W#16#500;
   STAT36[387] := W#16#1418;
   STAT36[388] := W#16#848;
   STAT36[389] := W#16#0;
   STAT36[390] := W#16#0;
   STAT36[391] := W#16#400;
   STAT36[392] := W#16#1418;
   STAT36[393] := W#16#848;
   STAT36[394] := W#16#0;
   STAT36[395] := W#16#0;
   STAT36[396] := W#16#500;
   STAT36[397] := W#16#1418;
   STAT36[398] := W#16#846;
   STAT36[399] := W#16#0;
   STAT36[400] := W#16#0;
   STAT36[401] := W#16#400;
   STAT36[402] := W#16#1418;
   STAT36[403] := W#16#749;
   STAT36[404] := W#16#0;
   STAT36[405] := W#16#2695;
   STAT36[406] := W#16#300;
   STAT36[407] := W#16#1418;
   STAT36[408] := W#16#746;
   STAT36[409] := W#16#B;
   STAT36[410] := W#16#2691;
   STAT36[411] := W#16#200;
   STAT36[412] := W#16#1418;
   STAT36[413] := W#16#744;
   STAT36[414] := W#16#1;
   STAT36[415] := W#16#0;
   STAT36[416] := W#16#500;
   STAT36[417] := W#16#1418;
   STAT36[418] := W#16#735;
   STAT36[419] := W#16#0;
   STAT36[420] := W#16#0;
   STAT36[421] := W#16#400;
   STAT36[422] := W#16#1418;
   STAT36[423] := W#16#735;
   STAT36[424] := W#16#0;
   STAT36[425] := W#16#0;
   STAT36[426] := W#16#500;
   STAT36[427] := W#16#1418;
   STAT36[428] := W#16#734;
   STAT36[429] := W#16#0;
   STAT36[430] := W#16#0;
   STAT36[431] := W#16#400;
   STAT36[432] := W#16#1418;
   STAT36[433] := W#16#634;
   STAT36[434] := W#16#0;
   STAT36[435] := W#16#2694;
   STAT36[436] := W#16#300;
   STAT36[437] := W#16#1418;
   STAT36[438] := W#16#632;
   STAT36[439] := W#16#B;
   STAT36[440] := W#16#2690;
   STAT36[441] := W#16#200;
   STAT36[442] := W#16#1418;
   STAT36[443] := W#16#630;
   STAT36[444] := W#16#1;
   STAT36[445] := W#16#0;
   STAT36[446] := W#16#500;
   STAT36[447] := W#16#1418;
   STAT36[448] := W#16#621;
   STAT36[449] := W#16#0;
   STAT36[450] := W#16#0;
   STAT36[451] := W#16#400;
   STAT36[452] := W#16#1418;
   STAT36[453] := W#16#620;
   STAT36[454] := W#16#0;
   STAT36[455] := W#16#0;
   STAT36[456] := W#16#500;
   STAT36[457] := W#16#1418;
   STAT36[458] := W#16#619;
   STAT36[459] := W#16#0;
   STAT36[460] := W#16#0;
   STAT36[461] := W#16#400;
   STAT36[462] := W#16#1418;
   STAT36[463] := W#16#228;
   STAT36[464] := W#16#0;
   STAT36[465] := W#16#2693;
   STAT36[466] := W#16#300;
   STAT36[467] := W#16#1418;
   STAT36[468] := W#16#226;
   STAT36[469] := W#16#B;
   STAT36[470] := W#16#2689;
   STAT36[471] := W#16#200;
   STAT36[472] := W#16#1418;
   STAT36[473] := W#16#224;
   STAT36[474] := W#16#1;
   STAT36[475] := W#16#0;
   STAT36[476] := W#16#500;
   STAT36[477] := W#16#1418;
   STAT36[478] := W#16#215;
   STAT36[479] := W#16#0;
   STAT36[480] := W#16#0;
   STAT36[481] := W#16#400;
   STAT36[482] := W#16#1418;
   STAT36[483] := W#16#215;
   STAT36[484] := W#16#0;
   STAT36[485] := W#16#0;
   STAT36[486] := W#16#500;
   STAT36[487] := W#16#1418;
   STAT36[488] := W#16#213;
   STAT36[489] := W#16#0;
   STAT36[490] := W#16#0;
   STAT36[491] := W#16#400;
   STAT36[492] := W#16#1418;
   STAT36[493] := W#16#115;
   STAT36[494] := W#16#0;
   STAT36[495] := W#16#2692;
   STAT36[496] := W#16#300;
   STAT36[497] := W#16#1418;
   STAT36[498] := W#16#112;
   STAT36[499] := W#16#B;
   STAT36[500] := W#16#2688;
   STAT37[1] := B#16#0;
   STAT37[2] := B#16#87;
   STAT37[3] := B#16#27;
   STAT37[4] := B#16#5;
   STAT37[5] := B#16#22;
   STAT37[6] := B#16#A;
   STAT37[7] := B#16#80;
   STAT37[8] := B#16#10;
   STAT37[9] := B#16#26;
   STAT37[10] := B#16#10;
   STAT37[11] := B#16#40;
   STAT37[12] := B#16#0;
   STAT37[13] := B#16#0;
   STAT37[14] := B#16#0;
   STAT37[15] := B#16#0;
   STAT37[16] := B#16#0;
   STAT38[1] := B#16#0;
   STAT38[2] := B#16#0;
   STAT38[3] := B#16#0;
   STAT38[4] := B#16#0;
   STAT39[1] := B#16#27;
   STAT39[2] := B#16#9;
   STAT39[3] := B#16#0;
   STAT39[4] := B#16#87;
   STAT39[5] := B#16#A;
   STAT39[6] := B#16#22;
   STAT39[7] := B#16#10;
   STAT39[8] := B#16#80;
   STAT39[9] := B#16#10;
   STAT39[10] := B#16#16;
   STAT39[11] := B#16#0;
   STAT39[12] := B#16#40;
   STAT39[13] := B#16#0;
   STAT39[14] := B#16#0;
   STAT39[15] := B#16#0;
   STAT39[16] := B#16#0;
END_DATA_BLOCK

DATA_BLOCK DB 170
VERSION : 0.1


  STRUCT
   STAT0 : WORD ;
   STAT1 : WORD ;
   STAT2 : WORD ;
   STAT3 : WORD ;
   STAT4 : WORD ;
   STAT5 : WORD ;
   STAT6 : WORD ;
   STAT7 : WORD ;
   STAT8 : WORD ;
   STAT9 : WORD ;
   STAT10 : WORD ;
   STAT11 : WORD ;
   STAT12 : WORD ;
   STAT13 : WORD ;
   STAT14 : WORD ;
   STAT15 : WORD ;
   STAT16 : INT ;
   STAT17 : INT ;
   STAT18 : INT ;
   STAT19 : INT ;
   STAT20 : ARRAY  [1 .. 6 ] OF BYTE ;
   STAT21 : ARRAY  [1 .. 6 ] OF BYTE ;
   STAT22 : ARRAY  [1 .. 40 ] OF BOOL  := FALSE;
   STAT23 : ARRAY  [1 .. 40 ] OF BOOL  := FALSE;
   STAT24 : WORD ;
   STAT25 : WORD ;
   STAT26 : WORD ;
   STAT27 : WORD ;
   STAT28 : WORD ;
   STAT29 : WORD ;
   STAT30 : WORD ;
   STAT31 : ARRAY  [1 .. 7 ] OF WORD ;
   STAT32 : INT ;
   STAT33 : INT ;
   STAT34 : INT ;
   STAT35 : INT ;
   STAT36 : ARRAY  [1 .. 500 ] OF WORD ;
   STAT37 : ARRAY  [1 .. 16 ] OF BYTE ;
   STAT38 : ARRAY  [1 .. 4 ] OF BYTE ;
   STAT39 : ARRAY  [1 .. 16 ] OF BYTE ;
  END_STRUCT ;
BEGIN
   STAT0 := W#16#0;
   STAT1 := W#16#0;
   STAT2 := W#16#0;
   STAT3 := W#16#0;
   STAT4 := W#16#0;
   STAT5 := W#16#0;
   STAT6 := W#16#0;
   STAT7 := W#16#0;
   STAT8 := W#16#0;
   STAT9 := W#16#0;
   STAT10 := W#16#0;
   STAT11 := W#16#0;
   STAT12 := W#16#0;
   STAT13 := W#16#0;
   STAT14 := W#16#0;
   STAT15 := W#16#0;
   STAT16 := 0;
   STAT17 := 0;
   STAT18 := 0;
   STAT19 := 0;
   STAT20[1] := B#16#0;
   STAT20[2] := B#16#0;
   STAT20[3] := B#16#0;
   STAT20[4] := B#16#0;
   STAT20[5] := B#16#0;
   STAT20[6] := B#16#0;
   STAT21[1] := B#16#0;
   STAT21[2] := B#16#0;
   STAT21[3] := B#16#0;
   STAT21[4] := B#16#0;
   STAT21[5] := B#16#0;
   STAT21[6] := B#16#0;
   STAT22[1] := FALSE;
   STAT22[2] := FALSE;
   STAT22[3] := FALSE;
   STAT22[4] := FALSE;
   STAT22[5] := FALSE;
   STAT22[6] := FALSE;
   STAT22[7] := FALSE;
   STAT22[8] := FALSE;
   STAT22[9] := FALSE;
   STAT22[10] := FALSE;
   STAT22[11] := FALSE;
   STAT22[12] := FALSE;
   STAT22[13] := FALSE;
   STAT22[14] := FALSE;
   STAT22[15] := FALSE;
   STAT22[16] := FALSE;
   STAT22[17] := FALSE;
   STAT22[18] := FALSE;
   STAT22[19] := FALSE;
   STAT22[20] := FALSE;
   STAT22[21] := FALSE;
   STAT22[22] := FALSE;
   STAT22[23] := FALSE;
   STAT22[24] := FALSE;
   STAT22[25] := FALSE;
   STAT22[26] := FALSE;
   STAT22[27] := FALSE;
   STAT22[28] := FALSE;
   STAT22[29] := FALSE;
   STAT22[30] := FALSE;
   STAT22[31] := FALSE;
   STAT22[32] := FALSE;
   STAT22[33] := FALSE;
   STAT22[34] := FALSE;
   STAT22[35] := FALSE;
   STAT22[36] := FALSE;
   STAT22[37] := FALSE;
   STAT22[38] := FALSE;
   STAT22[39] := FALSE;
   STAT22[40] := FALSE;
   STAT23[1] := FALSE;
   STAT23[2] := FALSE;
   STAT23[3] := FALSE;
   STAT23[4] := FALSE;
   STAT23[5] := FALSE;
   STAT23[6] := FALSE;
   STAT23[7] := FALSE;
   STAT23[8] := FALSE;
   STAT23[9] := FALSE;
   STAT23[10] := FALSE;
   STAT23[11] := FALSE;
   STAT23[12] := FALSE;
   STAT23[13] := FALSE;
   STAT23[14] := FALSE;
   STAT23[15] := FALSE;
   STAT23[16] := FALSE;
   STAT23[17] := FALSE;
   STAT23[18] := FALSE;
   STAT23[19] := FALSE;
   STAT23[20] := FALSE;
   STAT23[21] := FALSE;
   STAT23[22] := FALSE;
   STAT23[23] := FALSE;
   STAT23[24] := FALSE;
   STAT23[25] := FALSE;
   STAT23[26] := FALSE;
   STAT23[27] := FALSE;
   STAT23[28] := FALSE;
   STAT23[29] := FALSE;
   STAT23[30] := FALSE;
   STAT23[31] := FALSE;
   STAT23[32] := FALSE;
   STAT23[33] := FALSE;
   STAT23[34] := FALSE;
   STAT23[35] := FALSE;
   STAT23[36] := FALSE;
   STAT23[37] := FALSE;
   STAT23[38] := FALSE;
   STAT23[39] := FALSE;
   STAT23[40] := FALSE;
   STAT24 := W#16#0;
   STAT25 := W#16#0;
   STAT26 := W#16#0;
   STAT27 := W#16#0;
   STAT28 := W#16#0;
   STAT29 := W#16#0;
   STAT30 := W#16#0;
   STAT31[1] := W#16#0;
   STAT31[2] := W#16#0;
   STAT31[3] := W#16#0;
   STAT31[4] := W#16#0;
   STAT31[5] := W#16#0;
   STAT31[6] := W#16#0;
   STAT31[7] := W#16#0;
   STAT32 := 0;
   STAT33 := 0;
   STAT34 := 0;
   STAT35 := 0;
   STAT36[1] := W#16#0;
   STAT36[2] := W#16#0;
   STAT36[3] := W#16#0;
   STAT36[4] := W#16#0;
   STAT36[5] := W#16#0;
   STAT36[6] := W#16#0;
   STAT36[7] := W#16#0;
   STAT36[8] := W#16#0;
   STAT36[9] := W#16#0;
   STAT36[10] := W#16#0;
   STAT36[11] := W#16#0;
   STAT36[12] := W#16#0;
   STAT36[13] := W#16#0;
   STAT36[14] := W#16#0;
   STAT36[15] := W#16#0;
   STAT36[16] := W#16#0;
   STAT36[17] := W#16#0;
   STAT36[18] := W#16#0;
   STAT36[19] := W#16#0;
   STAT36[20] := W#16#0;
   STAT36[21] := W#16#0;
   STAT36[22] := W#16#0;
   STAT36[23] := W#16#0;
   STAT36[24] := W#16#0;
   STAT36[25] := W#16#0;
   STAT36[26] := W#16#0;
   STAT36[27] := W#16#0;
   STAT36[28] := W#16#0;
   STAT36[29] := W#16#0;
   STAT36[30] := W#16#0;
   STAT36[31] := W#16#0;
   STAT36[32] := W#16#0;
   STAT36[33] := W#16#0;
   STAT36[34] := W#16#0;
   STAT36[35] := W#16#0;
   STAT36[36] := W#16#0;
   STAT36[37] := W#16#0;
   STAT36[38] := W#16#0;
   STAT36[39] := W#16#0;
   STAT36[40] := W#16#0;
   STAT36[41] := W#16#0;
   STAT36[42] := W#16#0;
   STAT36[43] := W#16#0;
   STAT36[44] := W#16#0;
   STAT36[45] := W#16#0;
   STAT36[46] := W#16#0;
   STAT36[47] := W#16#0;
   STAT36[48] := W#16#0;
   STAT36[49] := W#16#0;
   STAT36[50] := W#16#0;
   STAT36[51] := W#16#0;
   STAT36[52] := W#16#0;
   STAT36[53] := W#16#0;
   STAT36[54] := W#16#0;
   STAT36[55] := W#16#0;
   STAT36[56] := W#16#0;
   STAT36[57] := W#16#0;
   STAT36[58] := W#16#0;
   STAT36[59] := W#16#0;
   STAT36[60] := W#16#0;
   STAT36[61] := W#16#0;
   STAT36[62] := W#16#0;
   STAT36[63] := W#16#0;
   STAT36[64] := W#16#0;
   STAT36[65] := W#16#0;
   STAT36[66] := W#16#0;
   STAT36[67] := W#16#0;
   STAT36[68] := W#16#0;
   STAT36[69] := W#16#0;
   STAT36[70] := W#16#0;
   STAT36[71] := W#16#0;
   STAT36[72] := W#16#0;
   STAT36[73] := W#16#0;
   STAT36[74] := W#16#0;
   STAT36[75] := W#16#0;
   STAT36[76] := W#16#0;
   STAT36[77] := W#16#0;
   STAT36[78] := W#16#0;
   STAT36[79] := W#16#0;
   STAT36[80] := W#16#0;
   STAT36[81] := W#16#0;
   STAT36[82] := W#16#0;
   STAT36[83] := W#16#0;
   STAT36[84] := W#16#0;
   STAT36[85] := W#16#0;
   STAT36[86] := W#16#0;
   STAT36[87] := W#16#0;
   STAT36[88] := W#16#0;
   STAT36[89] := W#16#0;
   STAT36[90] := W#16#0;
   STAT36[91] := W#16#0;
   STAT36[92] := W#16#0;
   STAT36[93] := W#16#0;
   STAT36[94] := W#16#0;
   STAT36[95] := W#16#0;
   STAT36[96] := W#16#0;
   STAT36[97] := W#16#0;
   STAT36[98] := W#16#0;
   STAT36[99] := W#16#0;
   STAT36[100] := W#16#0;
   STAT36[101] := W#16#0;
   STAT36[102] := W#16#0;
   STAT36[103] := W#16#0;
   STAT36[104] := W#16#0;
   STAT36[105] := W#16#0;
   STAT36[106] := W#16#0;
   STAT36[107] := W#16#0;
   STAT36[108] := W#16#0;
   STAT36[109] := W#16#0;
   STAT36[110] := W#16#0;
   STAT36[111] := W#16#0;
   STAT36[112] := W#16#0;
   STAT36[113] := W#16#0;
   STAT36[114] := W#16#0;
   STAT36[115] := W#16#0;
   STAT36[116] := W#16#0;
   STAT36[117] := W#16#0;
   STAT36[118] := W#16#0;
   STAT36[119] := W#16#0;
   STAT36[120] := W#16#0;
   STAT36[121] := W#16#0;
   STAT36[122] := W#16#0;
   STAT36[123] := W#16#0;
   STAT36[124] := W#16#0;
   STAT36[125] := W#16#0;
   STAT36[126] := W#16#0;
   STAT36[127] := W#16#0;
   STAT36[128] := W#16#0;
   STAT36[129] := W#16#0;
   STAT36[130] := W#16#0;
   STAT36[131] := W#16#0;
   STAT36[132] := W#16#0;
   STAT36[133] := W#16#0;
   STAT36[134] := W#16#0;
   STAT36[135] := W#16#0;
   STAT36[136] := W#16#0;
   STAT36[137] := W#16#0;
   STAT36[138] := W#16#0;
   STAT36[139] := W#16#0;
   STAT36[140] := W#16#0;
   STAT36[141] := W#16#0;
   STAT36[142] := W#16#0;
   STAT36[143] := W#16#0;
   STAT36[144] := W#16#0;
   STAT36[145] := W#16#0;
   STAT36[146] := W#16#0;
   STAT36[147] := W#16#0;
   STAT36[148] := W#16#0;
   STAT36[149] := W#16#0;
   STAT36[150] := W#16#0;
   STAT36[151] := W#16#0;
   STAT36[152] := W#16#0;
   STAT36[153] := W#16#0;
   STAT36[154] := W#16#0;
   STAT36[155] := W#16#0;
   STAT36[156] := W#16#0;
   STAT36[157] := W#16#0;
   STAT36[158] := W#16#0;
   STAT36[159] := W#16#0;
   STAT36[160] := W#16#0;
   STAT36[161] := W#16#0;
   STAT36[162] := W#16#0;
   STAT36[163] := W#16#0;
   STAT36[164] := W#16#0;
   STAT36[165] := W#16#0;
   STAT36[166] := W#16#0;
   STAT36[167] := W#16#0;
   STAT36[168] := W#16#0;
   STAT36[169] := W#16#0;
   STAT36[170] := W#16#0;
   STAT36[171] := W#16#0;
   STAT36[172] := W#16#0;
   STAT36[173] := W#16#0;
   STAT36[174] := W#16#0;
   STAT36[175] := W#16#0;
   STAT36[176] := W#16#0;
   STAT36[177] := W#16#0;
   STAT36[178] := W#16#0;
   STAT36[179] := W#16#0;
   STAT36[180] := W#16#0;
   STAT36[181] := W#16#0;
   STAT36[182] := W#16#0;
   STAT36[183] := W#16#0;
   STAT36[184] := W#16#0;
   STAT36[185] := W#16#0;
   STAT36[186] := W#16#0;
   STAT36[187] := W#16#0;
   STAT36[188] := W#16#0;
   STAT36[189] := W#16#0;
   STAT36[190] := W#16#0;
   STAT36[191] := W#16#0;
   STAT36[192] := W#16#0;
   STAT36[193] := W#16#0;
   STAT36[194] := W#16#0;
   STAT36[195] := W#16#0;
   STAT36[196] := W#16#0;
   STAT36[197] := W#16#0;
   STAT36[198] := W#16#0;
   STAT36[199] := W#16#0;
   STAT36[200] := W#16#0;
   STAT36[201] := W#16#0;
   STAT36[202] := W#16#0;
   STAT36[203] := W#16#0;
   STAT36[204] := W#16#0;
   STAT36[205] := W#16#0;
   STAT36[206] := W#16#0;
   STAT36[207] := W#16#0;
   STAT36[208] := W#16#0;
   STAT36[209] := W#16#0;
   STAT36[210] := W#16#0;
   STAT36[211] := W#16#0;
   STAT36[212] := W#16#0;
   STAT36[213] := W#16#0;
   STAT36[214] := W#16#0;
   STAT36[215] := W#16#0;
   STAT36[216] := W#16#0;
   STAT36[217] := W#16#0;
   STAT36[218] := W#16#0;
   STAT36[219] := W#16#0;
   STAT36[220] := W#16#0;
   STAT36[221] := W#16#0;
   STAT36[222] := W#16#0;
   STAT36[223] := W#16#0;
   STAT36[224] := W#16#0;
   STAT36[225] := W#16#0;
   STAT36[226] := W#16#0;
   STAT36[227] := W#16#0;
   STAT36[228] := W#16#0;
   STAT36[229] := W#16#0;
   STAT36[230] := W#16#0;
   STAT36[231] := W#16#0;
   STAT36[232] := W#16#0;
   STAT36[233] := W#16#0;
   STAT36[234] := W#16#0;
   STAT36[235] := W#16#0;
   STAT36[236] := W#16#0;
   STAT36[237] := W#16#0;
   STAT36[238] := W#16#0;
   STAT36[239] := W#16#0;
   STAT36[240] := W#16#0;
   STAT36[241] := W#16#0;
   STAT36[242] := W#16#0;
   STAT36[243] := W#16#0;
   STAT36[244] := W#16#0;
   STAT36[245] := W#16#0;
   STAT36[246] := W#16#0;
   STAT36[247] := W#16#0;
   STAT36[248] := W#16#0;
   STAT36[249] := W#16#0;
   STAT36[250] := W#16#0;
   STAT36[251] := W#16#0;
   STAT36[252] := W#16#0;
   STAT36[253] := W#16#0;
   STAT36[254] := W#16#0;
   STAT36[255] := W#16#0;
   STAT36[256] := W#16#0;
   STAT36[257] := W#16#0;
   STAT36[258] := W#16#0;
   STAT36[259] := W#16#0;
   STAT36[260] := W#16#0;
   STAT36[261] := W#16#0;
   STAT36[262] := W#16#0;
   STAT36[263] := W#16#0;
   STAT36[264] := W#16#0;
   STAT36[265] := W#16#0;
   STAT36[266] := W#16#0;
   STAT36[267] := W#16#0;
   STAT36[268] := W#16#0;
   STAT36[269] := W#16#0;
   STAT36[270] := W#16#0;
   STAT36[271] := W#16#0;
   STAT36[272] := W#16#0;
   STAT36[273] := W#16#0;
   STAT36[274] := W#16#0;
   STAT36[275] := W#16#0;
   STAT36[276] := W#16#0;
   STAT36[277] := W#16#0;
   STAT36[278] := W#16#0;
   STAT36[279] := W#16#0;
   STAT36[280] := W#16#0;
   STAT36[281] := W#16#0;
   STAT36[282] := W#16#0;
   STAT36[283] := W#16#0;
   STAT36[284] := W#16#0;
   STAT36[285] := W#16#0;
   STAT36[286] := W#16#0;
   STAT36[287] := W#16#0;
   STAT36[288] := W#16#0;
   STAT36[289] := W#16#0;
   STAT36[290] := W#16#0;
   STAT36[291] := W#16#0;
   STAT36[292] := W#16#0;
   STAT36[293] := W#16#0;
   STAT36[294] := W#16#0;
   STAT36[295] := W#16#0;
   STAT36[296] := W#16#0;
   STAT36[297] := W#16#0;
   STAT36[298] := W#16#0;
   STAT36[299] := W#16#0;
   STAT36[300] := W#16#0;
   STAT36[301] := W#16#0;
   STAT36[302] := W#16#0;
   STAT36[303] := W#16#0;
   STAT36[304] := W#16#0;
   STAT36[305] := W#16#0;
   STAT36[306] := W#16#0;
   STAT36[307] := W#16#0;
   STAT36[308] := W#16#0;
   STAT36[309] := W#16#0;
   STAT36[310] := W#16#0;
   STAT36[311] := W#16#0;
   STAT36[312] := W#16#0;
   STAT36[313] := W#16#0;
   STAT36[314] := W#16#0;
   STAT36[315] := W#16#0;
   STAT36[316] := W#16#0;
   STAT36[317] := W#16#0;
   STAT36[318] := W#16#0;
   STAT36[319] := W#16#0;
   STAT36[320] := W#16#0;
   STAT36[321] := W#16#0;
   STAT36[322] := W#16#0;
   STAT36[323] := W#16#0;
   STAT36[324] := W#16#0;
   STAT36[325] := W#16#0;
   STAT36[326] := W#16#0;
   STAT36[327] := W#16#0;
   STAT36[328] := W#16#0;
   STAT36[329] := W#16#0;
   STAT36[330] := W#16#0;
   STAT36[331] := W#16#0;
   STAT36[332] := W#16#0;
   STAT36[333] := W#16#0;
   STAT36[334] := W#16#0;
   STAT36[335] := W#16#0;
   STAT36[336] := W#16#0;
   STAT36[337] := W#16#0;
   STAT36[338] := W#16#0;
   STAT36[339] := W#16#0;
   STAT36[340] := W#16#0;
   STAT36[341] := W#16#0;
   STAT36[342] := W#16#0;
   STAT36[343] := W#16#0;
   STAT36[344] := W#16#0;
   STAT36[345] := W#16#0;
   STAT36[346] := W#16#0;
   STAT36[347] := W#16#0;
   STAT36[348] := W#16#0;
   STAT36[349] := W#16#0;
   STAT36[350] := W#16#0;
   STAT36[351] := W#16#0;
   STAT36[352] := W#16#0;
   STAT36[353] := W#16#0;
   STAT36[354] := W#16#0;
   STAT36[355] := W#16#0;
   STAT36[356] := W#16#0;
   STAT36[357] := W#16#0;
   STAT36[358] := W#16#0;
   STAT36[359] := W#16#0;
   STAT36[360] := W#16#0;
   STAT36[361] := W#16#0;
   STAT36[362] := W#16#0;
   STAT36[363] := W#16#0;
   STAT36[364] := W#16#0;
   STAT36[365] := W#16#0;
   STAT36[366] := W#16#0;
   STAT36[367] := W#16#0;
   STAT36[368] := W#16#0;
   STAT36[369] := W#16#0;
   STAT36[370] := W#16#0;
   STAT36[371] := W#16#0;
   STAT36[372] := W#16#0;
   STAT36[373] := W#16#0;
   STAT36[374] := W#16#0;
   STAT36[375] := W#16#0;
   STAT36[376] := W#16#0;
   STAT36[377] := W#16#0;
   STAT36[378] := W#16#0;
   STAT36[379] := W#16#0;
   STAT36[380] := W#16#0;
   STAT36[381] := W#16#0;
   STAT36[382] := W#16#0;
   STAT36[383] := W#16#0;
   STAT36[384] := W#16#0;
   STAT36[385] := W#16#0;
   STAT36[386] := W#16#0;
   STAT36[387] := W#16#0;
   STAT36[388] := W#16#0;
   STAT36[389] := W#16#0;
   STAT36[390] := W#16#0;
   STAT36[391] := W#16#0;
   STAT36[392] := W#16#0;
   STAT36[393] := W#16#0;
   STAT36[394] := W#16#0;
   STAT36[395] := W#16#0;
   STAT36[396] := W#16#0;
   STAT36[397] := W#16#0;
   STAT36[398] := W#16#0;
   STAT36[399] := W#16#0;
   STAT36[400] := W#16#0;
   STAT36[401] := W#16#0;
   STAT36[402] := W#16#0;
   STAT36[403] := W#16#0;
   STAT36[404] := W#16#0;
   STAT36[405] := W#16#0;
   STAT36[406] := W#16#0;
   STAT36[407] := W#16#0;
   STAT36[408] := W#16#0;
   STAT36[409] := W#16#0;
   STAT36[410] := W#16#0;
   STAT36[411] := W#16#0;
   STAT36[412] := W#16#0;
   STAT36[413] := W#16#0;
   STAT36[414] := W#16#0;
   STAT36[415] := W#16#0;
   STAT36[416] := W#16#0;
   STAT36[417] := W#16#0;
   STAT36[418] := W#16#0;
   STAT36[419] := W#16#0;
   STAT36[420] := W#16#0;
   STAT36[421] := W#16#0;
   STAT36[422] := W#16#0;
   STAT36[423] := W#16#0;
   STAT36[424] := W#16#0;
   STAT36[425] := W#16#0;
   STAT36[426] := W#16#0;
   STAT36[427] := W#16#0;
   STAT36[428] := W#16#0;
   STAT36[429] := W#16#0;
   STAT36[430] := W#16#0;
   STAT36[431] := W#16#0;
   STAT36[432] := W#16#0;
   STAT36[433] := W#16#0;
   STAT36[434] := W#16#0;
   STAT36[435] := W#16#0;
   STAT36[436] := W#16#0;
   STAT36[437] := W#16#0;
   STAT36[438] := W#16#0;
   STAT36[439] := W#16#0;
   STAT36[440] := W#16#0;
   STAT36[441] := W#16#0;
   STAT36[442] := W#16#0;
   STAT36[443] := W#16#0;
   STAT36[444] := W#16#0;
   STAT36[445] := W#16#0;
   STAT36[446] := W#16#0;
   STAT36[447] := W#16#0;
   STAT36[448] := W#16#0;
   STAT36[449] := W#16#0;
   STAT36[450] := W#16#0;
   STAT36[451] := W#16#0;
   STAT36[452] := W#16#0;
   STAT36[453] := W#16#0;
   STAT36[454] := W#16#0;
   STAT36[455] := W#16#0;
   STAT36[456] := W#16#0;
   STAT36[457] := W#16#0;
   STAT36[458] := W#16#0;
   STAT36[459] := W#16#0;
   STAT36[460] := W#16#0;
   STAT36[461] := W#16#0;
   STAT36[462] := W#16#0;
   STAT36[463] := W#16#0;
   STAT36[464] := W#16#0;
   STAT36[465] := W#16#0;
   STAT36[466] := W#16#0;
   STAT36[467] := W#16#0;
   STAT36[468] := W#16#0;
   STAT36[469] := W#16#0;
   STAT36[470] := W#16#0;
   STAT36[471] := W#16#0;
   STAT36[472] := W#16#0;
   STAT36[473] := W#16#0;
   STAT36[474] := W#16#0;
   STAT36[475] := W#16#0;
   STAT36[476] := W#16#0;
   STAT36[477] := W#16#0;
   STAT36[478] := W#16#0;
   STAT36[479] := W#16#0;
   STAT36[480] := W#16#0;
   STAT36[481] := W#16#0;
   STAT36[482] := W#16#0;
   STAT36[483] := W#16#0;
   STAT36[484] := W#16#0;
   STAT36[485] := W#16#0;
   STAT36[486] := W#16#0;
   STAT36[487] := W#16#0;
   STAT36[488] := W#16#0;
   STAT36[489] := W#16#0;
   STAT36[490] := W#16#0;
   STAT36[491] := W#16#0;
   STAT36[492] := W#16#0;
   STAT36[493] := W#16#0;
   STAT36[494] := W#16#0;
   STAT36[495] := W#16#0;
   STAT36[496] := W#16#0;
   STAT36[497] := W#16#0;
   STAT36[498] := W#16#0;
   STAT36[499] := W#16#0;
   STAT36[500] := W#16#0;
   STAT37[1] := B#16#0;
   STAT37[2] := B#16#0;
   STAT37[3] := B#16#0;
   STAT37[4] := B#16#0;
   STAT37[5] := B#16#0;
   STAT37[6] := B#16#0;
   STAT37[7] := B#16#0;
   STAT37[8] := B#16#0;
   STAT37[9] := B#16#0;
   STAT37[10] := B#16#0;
   STAT37[11] := B#16#0;
   STAT37[12] := B#16#0;
   STAT37[13] := B#16#0;
   STAT37[14] := B#16#0;
   STAT37[15] := B#16#0;
   STAT37[16] := B#16#0;
   STAT38[1] := B#16#0;
   STAT38[2] := B#16#0;
   STAT38[3] := B#16#0;
   STAT38[4] := B#16#0;
   STAT39[1] := B#16#0;
   STAT39[2] := B#16#0;
   STAT39[3] := B#16#0;
   STAT39[4] := B#16#0;
   STAT39[5] := B#16#0;
   STAT39[6] := B#16#0;
   STAT39[7] := B#16#0;
   STAT39[8] := B#16#0;
   STAT39[9] := B#16#0;
   STAT39[10] := B#16#0;
   STAT39[11] := B#16#0;
   STAT39[12] := B#16#0;
   STAT39[13] := B#16#0;
   STAT39[14] := B#16#0;
   STAT39[15] := B#16#0;
   STAT39[16] := B#16#0;
END_DATA_BLOCK

DATA_BLOCK DB 171
VERSION : 0.1


  STRUCT
   STAT0 : ARRAY  [1 .. 320 ] OF BYTE ;
   STAT1 : INT ;
   STAT2 : WORD ;
   STAT3 : INT ;
   STAT4 : INT ;
   STAT5 : INT ;
   STAT6 : INT ;
   STAT7 : INT ;
   STAT8 : INT ;
   STAT9 : INT ;
   STAT10 : INT ;
   STAT11 : INT ;
   STAT12 : INT ;
   STAT13 : INT ;
   STAT14 : INT ;
   STAT15 : INT ;
   STAT16 : INT ;
   STAT17 : INT ;
   STAT18 : INT ;
   STAT19 : INT ;
   STAT20 : INT ;
   STAT21 : ARRAY  [1 .. 20 ] OF WORD ;
  END_STRUCT ;
BEGIN
   STAT0[1] := B#16#0;
   STAT0[2] := B#16#87;
   STAT0[3] := B#16#27;
   STAT0[4] := B#16#16;
   STAT0[5] := B#16#22;
   STAT0[6] := B#16#22;
   STAT0[7] := B#16#80;
   STAT0[8] := B#16#4;
   STAT0[9] := B#16#16;
   STAT0[10] := B#16#10;
   STAT0[11] := B#16#60;
   STAT0[12] := B#16#0;
   STAT0[13] := B#16#0;
   STAT0[14] := B#16#0;
   STAT0[15] := B#16#0;
   STAT0[16] := B#16#0;
   STAT0[17] := B#16#0;
   STAT0[18] := B#16#87;
   STAT0[19] := B#16#27;
   STAT0[20] := B#16#15;
   STAT0[21] := B#16#22;
   STAT0[22] := B#16#22;
   STAT0[23] := B#16#80;
   STAT0[24] := B#16#1;
   STAT0[25] := B#16#62;
   STAT0[26] := B#16#54;
   STAT0[27] := B#16#60;
   STAT0[28] := B#16#0;
   STAT0[29] := B#16#0;
   STAT0[30] := B#16#0;
   STAT0[31] := B#16#0;
   STAT0[32] := B#16#0;
   STAT0[33] := B#16#0;
   STAT0[34] := B#16#87;
   STAT0[35] := B#16#27;
   STAT0[36] := B#16#14;
   STAT0[37] := B#16#22;
   STAT0[38] := B#16#22;
   STAT0[39] := B#16#80;
   STAT0[40] := B#16#1;
   STAT0[41] := B#16#16;
   STAT0[42] := B#16#54;
   STAT0[43] := B#16#60;
   STAT0[44] := B#16#0;
   STAT0[45] := B#16#0;
   STAT0[46] := B#16#0;
   STAT0[47] := B#16#0;
   STAT0[48] := B#16#0;
   STAT0[49] := B#16#0;
   STAT0[50] := B#16#87;
   STAT0[51] := B#16#27;
   STAT0[52] := B#16#13;
   STAT0[53] := B#16#22;
   STAT0[54] := B#16#A;
   STAT0[55] := B#16#80;
   STAT0[56] := B#16#10;
   STAT0[57] := B#16#52;
   STAT0[58] := B#16#54;
   STAT0[59] := B#16#40;
   STAT0[60] := B#16#0;
   STAT0[61] := B#16#0;
   STAT0[62] := B#16#0;
   STAT0[63] := B#16#0;
   STAT0[64] := B#16#0;
   STAT0[65] := B#16#0;
   STAT0[66] := B#16#87;
   STAT0[67] := B#16#27;
   STAT0[68] := B#16#12;
   STAT0[69] := B#16#22;
   STAT0[70] := B#16#22;
   STAT0[71] := B#16#80;
   STAT0[72] := B#16#1;
   STAT0[73] := B#16#26;
   STAT0[74] := B#16#54;
   STAT0[75] := B#16#60;
   STAT0[76] := B#16#0;
   STAT0[77] := B#16#0;
   STAT0[78] := B#16#0;
   STAT0[79] := B#16#0;
   STAT0[80] := B#16#0;
   STAT0[81] := B#16#0;
   STAT0[82] := B#16#87;
   STAT0[83] := B#16#27;
   STAT0[84] := B#16#11;
   STAT0[85] := B#16#22;
   STAT0[86] := B#16#84;
   STAT0[87] := B#16#80;
   STAT0[88] := B#16#1;
   STAT0[89] := B#16#62;
   STAT0[90] := B#16#54;
   STAT0[91] := B#16#40;
   STAT0[92] := B#16#0;
   STAT0[93] := B#16#0;
   STAT0[94] := B#16#0;
   STAT0[95] := B#16#0;
   STAT0[96] := B#16#0;
   STAT0[97] := B#16#0;
   STAT0[98] := B#16#87;
   STAT0[99] := B#16#27;
   STAT0[100] := B#16#10;
   STAT0[101] := B#16#22;
   STAT0[102] := B#16#22;
   STAT0[103] := B#16#80;
   STAT0[104] := B#16#1;
   STAT0[105] := B#16#52;
   STAT0[106] := B#16#54;
   STAT0[107] := B#16#60;
   STAT0[108] := B#16#0;
   STAT0[109] := B#16#0;
   STAT0[110] := B#16#0;
   STAT0[111] := B#16#0;
   STAT0[112] := B#16#0;
   STAT0[113] := B#16#0;
   STAT0[114] := B#16#87;
   STAT0[115] := B#16#27;
   STAT0[116] := B#16#9;
   STAT0[117] := B#16#22;
   STAT0[118] := B#16#A;
   STAT0[119] := B#16#80;
   STAT0[120] := B#16#10;
   STAT0[121] := B#16#16;
   STAT0[122] := B#16#10;
   STAT0[123] := B#16#40;
   STAT0[124] := B#16#0;
   STAT0[125] := B#16#0;
   STAT0[126] := B#16#0;
   STAT0[127] := B#16#0;
   STAT0[128] := B#16#0;
   STAT0[129] := B#16#0;
   STAT0[130] := B#16#0;
   STAT0[131] := B#16#0;
   STAT0[132] := B#16#0;
   STAT0[133] := B#16#0;
   STAT0[134] := B#16#0;
   STAT0[135] := B#16#0;
   STAT0[136] := B#16#0;
   STAT0[137] := B#16#0;
   STAT0[138] := B#16#0;
   STAT0[139] := B#16#0;
   STAT0[140] := B#16#0;
   STAT0[141] := B#16#0;
   STAT0[142] := B#16#0;
   STAT0[143] := B#16#0;
   STAT0[144] := B#16#0;
   STAT0[145] := B#16#0;
   STAT0[146] := B#16#0;
   STAT0[147] := B#16#0;
   STAT0[148] := B#16#0;
   STAT0[149] := B#16#0;
   STAT0[150] := B#16#0;
   STAT0[151] := B#16#0;
   STAT0[152] := B#16#0;
   STAT0[153] := B#16#0;
   STAT0[154] := B#16#0;
   STAT0[155] := B#16#0;
   STAT0[156] := B#16#0;
   STAT0[157] := B#16#0;
   STAT0[158] := B#16#0;
   STAT0[159] := B#16#0;
   STAT0[160] := B#16#0;
   STAT0[161] := B#16#0;
   STAT0[162] := B#16#0;
   STAT0[163] := B#16#0;
   STAT0[164] := B#16#0;
   STAT0[165] := B#16#0;
   STAT0[166] := B#16#0;
   STAT0[167] := B#16#0;
   STAT0[168] := B#16#0;
   STAT0[169] := B#16#0;
   STAT0[170] := B#16#0;
   STAT0[171] := B#16#0;
   STAT0[172] := B#16#0;
   STAT0[173] := B#16#0;
   STAT0[174] := B#16#0;
   STAT0[175] := B#16#0;
   STAT0[176] := B#16#0;
   STAT0[177] := B#16#0;
   STAT0[178] := B#16#0;
   STAT0[179] := B#16#0;
   STAT0[180] := B#16#0;
   STAT0[181] := B#16#0;
   STAT0[182] := B#16#0;
   STAT0[183] := B#16#0;
   STAT0[184] := B#16#0;
   STAT0[185] := B#16#0;
   STAT0[186] := B#16#0;
   STAT0[187] := B#16#0;
   STAT0[188] := B#16#0;
   STAT0[189] := B#16#0;
   STAT0[190] := B#16#0;
   STAT0[191] := B#16#0;
   STAT0[192] := B#16#0;
   STAT0[193] := B#16#0;
   STAT0[194] := B#16#0;
   STAT0[195] := B#16#0;
   STAT0[196] := B#16#0;
   STAT0[197] := B#16#0;
   STAT0[198] := B#16#0;
   STAT0[199] := B#16#0;
   STAT0[200] := B#16#0;
   STAT0[201] := B#16#0;
   STAT0[202] := B#16#4;
   STAT0[203] := B#16#0;
   STAT0[204] := B#16#B;
   STAT0[205] := B#16#0;
   STAT0[206] := B#16#0;
   STAT0[207] := B#16#0;
   STAT0[208] := B#16#0;
   STAT0[209] := B#16#0;
   STAT0[210] := B#16#0;
   STAT0[211] := B#16#0;
   STAT0[212] := B#16#0;
   STAT0[213] := B#16#0;
   STAT0[214] := B#16#0;
   STAT0[215] := B#16#0;
   STAT0[216] := B#16#0;
   STAT0[217] := B#16#0;
   STAT0[218] := B#16#0;
   STAT0[219] := B#16#0;
   STAT0[220] := B#16#0;
   STAT0[221] := B#16#0;
   STAT0[222] := B#16#0;
   STAT0[223] := B#16#0;
   STAT0[224] := B#16#0;
   STAT0[225] := B#16#0;
   STAT0[226] := B#16#0;
   STAT0[227] := B#16#0;
   STAT0[228] := B#16#0;
   STAT0[229] := B#16#0;
   STAT0[230] := B#16#0;
   STAT0[231] := B#16#0;
   STAT0[232] := B#16#0;
   STAT0[233] := B#16#0;
   STAT0[234] := B#16#0;
   STAT0[235] := B#16#0;
   STAT0[236] := B#16#0;
   STAT0[237] := B#16#0;
   STAT0[238] := B#16#0;
   STAT0[239] := B#16#0;
   STAT0[240] := B#16#0;
   STAT0[241] := B#16#0;
   STAT0[242] := B#16#0;
   STAT0[243] := B#16#0;
   STAT0[244] := B#16#0;
   STAT0[245] := B#16#0;
   STAT0[246] := B#16#0;
   STAT0[247] := B#16#0;
   STAT0[248] := B#16#0;
   STAT0[249] := B#16#0;
   STAT0[250] := B#16#0;
   STAT0[251] := B#16#0;
   STAT0[252] := B#16#0;
   STAT0[253] := B#16#0;
   STAT0[254] := B#16#0;
   STAT0[255] := B#16#0;
   STAT0[256] := B#16#0;
   STAT0[257] := B#16#0;
   STAT0[258] := B#16#0;
   STAT0[259] := B#16#0;
   STAT0[260] := B#16#0;
   STAT0[261] := B#16#0;
   STAT0[262] := B#16#0;
   STAT0[263] := B#16#0;
   STAT0[264] := B#16#0;
   STAT0[265] := B#16#0;
   STAT0[266] := B#16#0;
   STAT0[267] := B#16#0;
   STAT0[268] := B#16#0;
   STAT0[269] := B#16#0;
   STAT0[270] := B#16#0;
   STAT0[271] := B#16#0;
   STAT0[272] := B#16#0;
   STAT0[273] := B#16#0;
   STAT0[274] := B#16#0;
   STAT0[275] := B#16#0;
   STAT0[276] := B#16#0;
   STAT0[277] := B#16#0;
   STAT0[278] := B#16#0;
   STAT0[279] := B#16#0;
   STAT0[280] := B#16#0;
   STAT0[281] := B#16#0;
   STAT0[282] := B#16#0;
   STAT0[283] := B#16#0;
   STAT0[284] := B#16#0;
   STAT0[285] := B#16#0;
   STAT0[286] := B#16#0;
   STAT0[287] := B#16#0;
   STAT0[288] := B#16#0;
   STAT0[289] := B#16#0;
   STAT0[290] := B#16#0;
   STAT0[291] := B#16#0;
   STAT0[292] := B#16#0;
   STAT0[293] := B#16#0;
   STAT0[294] := B#16#0;
   STAT0[295] := B#16#0;
   STAT0[296] := B#16#0;
   STAT0[297] := B#16#0;
   STAT0[298] := B#16#0;
   STAT0[299] := B#16#0;
   STAT0[300] := B#16#0;
   STAT0[301] := B#16#0;
   STAT0[302] := B#16#0;
   STAT0[303] := B#16#0;
   STAT0[304] := B#16#0;
   STAT0[305] := B#16#0;
   STAT0[306] := B#16#0;
   STAT0[307] := B#16#0;
   STAT0[308] := B#16#0;
   STAT0[309] := B#16#0;
   STAT0[310] := B#16#0;
   STAT0[311] := B#16#0;
   STAT0[312] := B#16#0;
   STAT0[313] := B#16#0;
   STAT0[314] := B#16#0;
   STAT0[315] := B#16#0;
   STAT0[316] := B#16#0;
   STAT0[317] := B#16#0;
   STAT0[318] := B#16#0;
   STAT0[319] := B#16#0;
   STAT0[320] := B#16#0;
   STAT1 := 0;
   STAT2 := W#16#300;
   STAT3 := 0;
   STAT4 := 0;
   STAT5 := 0;
   STAT6 := 0;
   STAT7 := 0;
   STAT8 := 0;
   STAT9 := 42;
   STAT10 := 74;
   STAT11 := 1;
   STAT12 := 0;
   STAT13 := 0;
   STAT14 := 0;
   STAT15 := 0;
   STAT16 := 0;
   STAT17 := 0;
   STAT18 := 0;
   STAT19 := 0;
   STAT20 := 80;
   STAT21[1] := W#16#0;
   STAT21[2] := W#16#0;
   STAT21[3] := W#16#0;
   STAT21[4] := W#16#0;
   STAT21[5] := W#16#0;
   STAT21[6] := W#16#0;
   STAT21[7] := W#16#0;
   STAT21[8] := W#16#0;
   STAT21[9] := W#16#0;
   STAT21[10] := W#16#0;
   STAT21[11] := W#16#205;
   STAT21[12] := W#16#0;
   STAT21[13] := W#16#0;
   STAT21[14] := W#16#0;
   STAT21[15] := W#16#0;
   STAT21[16] := W#16#0;
   STAT21[17] := W#16#0;
   STAT21[18] := W#16#0;
   STAT21[19] := W#16#0;
   STAT21[20] := W#16#0;
END_DATA_BLOCK

DATA_BLOCK DB 241
VERSION : 0.1


  STRUCT
   STAT0 : WORD ;
   STAT1 : WORD ;
   STAT2 : WORD ;
   STAT3 : WORD ;
   STAT4 : WORD ;
   STAT5 : WORD ;
   STAT6 : WORD ;
   STAT7 : WORD ;
   STAT8 : WORD ;
   STAT9 : WORD ;
   STAT10 : WORD ;
   STAT11 : WORD ;
   STAT12 : WORD ;
   STAT13 : WORD ;
   STAT14 : WORD ;
   STAT15 : WORD ;
   STAT16 : INT ;
   STAT17 : INT ;
   STAT18 : INT ;
   STAT19 : INT ;
   STAT20 : ARRAY  [1 .. 6 ] OF BYTE ;
   STAT21 : ARRAY  [1 .. 6 ] OF BYTE ;
   STAT22 : ARRAY  [1 .. 40 ] OF BOOL  := FALSE;
   STAT23 : ARRAY  [1 .. 40 ] OF BOOL  := FALSE;
   STAT24 : WORD ;
   STAT25 : WORD ;
   STAT26 : WORD ;
   STAT27 : WORD ;
   STAT28 : WORD ;
   STAT29 : WORD ;
   STAT30 : WORD ;
   STAT31 : ARRAY  [1 .. 7 ] OF WORD ;
   STAT32 : INT ;
   STAT33 : INT ;
   STAT34 : INT ;
   STAT35 : INT ;
   STAT36 : ARRAY  [1 .. 500 ] OF WORD ;
   STAT37 : ARRAY  [1 .. 16 ] OF BYTE ;
   STAT38 : ARRAY  [1 .. 4 ] OF BYTE ;
   STAT39 : ARRAY  [1 .. 16 ] OF BYTE ;
  END_STRUCT ;
BEGIN
   STAT0 := W#16#0;
   STAT1 := W#16#0;
   STAT2 := W#16#0;
   STAT3 := W#16#0;
   STAT4 := W#16#0;
   STAT5 := W#16#0;
   STAT6 := W#16#0;
   STAT7 := W#16#0;
   STAT8 := W#16#0;
   STAT9 := W#16#0;
   STAT10 := W#16#0;
   STAT11 := W#16#0;
   STAT12 := W#16#0;
   STAT13 := W#16#0;
   STAT14 := W#16#0;
   STAT15 := W#16#0;
   STAT16 := 0;
   STAT17 := 0;
   STAT18 := 0;
   STAT19 := 0;
   STAT20[1] := B#16#0;
   STAT20[2] := B#16#0;
   STAT20[3] := B#16#0;
   STAT20[4] := B#16#0;
   STAT20[5] := B#16#0;
   STAT20[6] := B#16#0;
   STAT21[1] := B#16#0;
   STAT21[2] := B#16#0;
   STAT21[3] := B#16#0;
   STAT21[4] := B#16#0;
   STAT21[5] := B#16#0;
   STAT21[6] := B#16#0;
   STAT22[1] := FALSE;
   STAT22[2] := FALSE;
   STAT22[3] := FALSE;
   STAT22[4] := FALSE;
   STAT22[5] := FALSE;
   STAT22[6] := FALSE;
   STAT22[7] := FALSE;
   STAT22[8] := FALSE;
   STAT22[9] := FALSE;
   STAT22[10] := FALSE;
   STAT22[11] := FALSE;
   STAT22[12] := FALSE;
   STAT22[13] := FALSE;
   STAT22[14] := FALSE;
   STAT22[15] := FALSE;
   STAT22[16] := FALSE;
   STAT22[17] := FALSE;
   STAT22[18] := FALSE;
   STAT22[19] := FALSE;
   STAT22[20] := FALSE;
   STAT22[21] := FALSE;
   STAT22[22] := FALSE;
   STAT22[23] := FALSE;
   STAT22[24] := FALSE;
   STAT22[25] := FALSE;
   STAT22[26] := FALSE;
   STAT22[27] := FALSE;
   STAT22[28] := FALSE;
   STAT22[29] := FALSE;
   STAT22[30] := FALSE;
   STAT22[31] := FALSE;
   STAT22[32] := FALSE;
   STAT22[33] := FALSE;
   STAT22[34] := FALSE;
   STAT22[35] := FALSE;
   STAT22[36] := FALSE;
   STAT22[37] := FALSE;
   STAT22[38] := FALSE;
   STAT22[39] := FALSE;
   STAT22[40] := FALSE;
   STAT23[1] := FALSE;
   STAT23[2] := FALSE;
   STAT23[3] := FALSE;
   STAT23[4] := FALSE;
   STAT23[5] := FALSE;
   STAT23[6] := FALSE;
   STAT23[7] := FALSE;
   STAT23[8] := FALSE;
   STAT23[9] := FALSE;
   STAT23[10] := FALSE;
   STAT23[11] := FALSE;
   STAT23[12] := FALSE;
   STAT23[13] := FALSE;
   STAT23[14] := FALSE;
   STAT23[15] := FALSE;
   STAT23[16] := FALSE;
   STAT23[17] := FALSE;
   STAT23[18] := FALSE;
   STAT23[19] := FALSE;
   STAT23[20] := FALSE;
   STAT23[21] := FALSE;
   STAT23[22] := FALSE;
   STAT23[23] := FALSE;
   STAT23[24] := FALSE;
   STAT23[25] := FALSE;
   STAT23[26] := FALSE;
   STAT23[27] := FALSE;
   STAT23[28] := FALSE;
   STAT23[29] := FALSE;
   STAT23[30] := FALSE;
   STAT23[31] := FALSE;
   STAT23[32] := FALSE;
   STAT23[33] := FALSE;
   STAT23[34] := FALSE;
   STAT23[35] := FALSE;
   STAT23[36] := FALSE;
   STAT23[37] := FALSE;
   STAT23[38] := FALSE;
   STAT23[39] := FALSE;
   STAT23[40] := FALSE;
   STAT24 := W#16#0;
   STAT25 := W#16#0;
   STAT26 := W#16#0;
   STAT27 := W#16#0;
   STAT28 := W#16#0;
   STAT29 := W#16#0;
   STAT30 := W#16#0;
   STAT31[1] := W#16#0;
   STAT31[2] := W#16#0;
   STAT31[3] := W#16#0;
   STAT31[4] := W#16#0;
   STAT31[5] := W#16#0;
   STAT31[6] := W#16#0;
   STAT31[7] := W#16#0;
   STAT32 := 0;
   STAT33 := 0;
   STAT34 := 0;
   STAT35 := 0;
   STAT36[1] := W#16#0;
   STAT36[2] := W#16#0;
   STAT36[3] := W#16#0;
   STAT36[4] := W#16#0;
   STAT36[5] := W#16#0;
   STAT36[6] := W#16#0;
   STAT36[7] := W#16#0;
   STAT36[8] := W#16#0;
   STAT36[9] := W#16#0;
   STAT36[10] := W#16#0;
   STAT36[11] := W#16#0;
   STAT36[12] := W#16#0;
   STAT36[13] := W#16#0;
   STAT36[14] := W#16#0;
   STAT36[15] := W#16#0;
   STAT36[16] := W#16#0;
   STAT36[17] := W#16#0;
   STAT36[18] := W#16#0;
   STAT36[19] := W#16#0;
   STAT36[20] := W#16#0;
   STAT36[21] := W#16#0;
   STAT36[22] := W#16#0;
   STAT36[23] := W#16#0;
   STAT36[24] := W#16#0;
   STAT36[25] := W#16#0;
   STAT36[26] := W#16#0;
   STAT36[27] := W#16#0;
   STAT36[28] := W#16#0;
   STAT36[29] := W#16#0;
   STAT36[30] := W#16#0;
   STAT36[31] := W#16#0;
   STAT36[32] := W#16#0;
   STAT36[33] := W#16#0;
   STAT36[34] := W#16#0;
   STAT36[35] := W#16#0;
   STAT36[36] := W#16#0;
   STAT36[37] := W#16#0;
   STAT36[38] := W#16#0;
   STAT36[39] := W#16#0;
   STAT36[40] := W#16#0;
   STAT36[41] := W#16#0;
   STAT36[42] := W#16#0;
   STAT36[43] := W#16#0;
   STAT36[44] := W#16#0;
   STAT36[45] := W#16#0;
   STAT36[46] := W#16#0;
   STAT36[47] := W#16#0;
   STAT36[48] := W#16#0;
   STAT36[49] := W#16#0;
   STAT36[50] := W#16#0;
   STAT36[51] := W#16#0;
   STAT36[52] := W#16#0;
   STAT36[53] := W#16#0;
   STAT36[54] := W#16#0;
   STAT36[55] := W#16#0;
   STAT36[56] := W#16#0;
   STAT36[57] := W#16#0;
   STAT36[58] := W#16#0;
   STAT36[59] := W#16#0;
   STAT36[60] := W#16#0;
   STAT36[61] := W#16#0;
   STAT36[62] := W#16#0;
   STAT36[63] := W#16#0;
   STAT36[64] := W#16#0;
   STAT36[65] := W#16#0;
   STAT36[66] := W#16#0;
   STAT36[67] := W#16#0;
   STAT36[68] := W#16#0;
   STAT36[69] := W#16#0;
   STAT36[70] := W#16#0;
   STAT36[71] := W#16#0;
   STAT36[72] := W#16#0;
   STAT36[73] := W#16#0;
   STAT36[74] := W#16#0;
   STAT36[75] := W#16#0;
   STAT36[76] := W#16#0;
   STAT36[77] := W#16#0;
   STAT36[78] := W#16#0;
   STAT36[79] := W#16#0;
   STAT36[80] := W#16#0;
   STAT36[81] := W#16#0;
   STAT36[82] := W#16#0;
   STAT36[83] := W#16#0;
   STAT36[84] := W#16#0;
   STAT36[85] := W#16#0;
   STAT36[86] := W#16#0;
   STAT36[87] := W#16#0;
   STAT36[88] := W#16#0;
   STAT36[89] := W#16#0;
   STAT36[90] := W#16#0;
   STAT36[91] := W#16#0;
   STAT36[92] := W#16#0;
   STAT36[93] := W#16#0;
   STAT36[94] := W#16#0;
   STAT36[95] := W#16#0;
   STAT36[96] := W#16#0;
   STAT36[97] := W#16#0;
   STAT36[98] := W#16#0;
   STAT36[99] := W#16#0;
   STAT36[100] := W#16#0;
   STAT36[101] := W#16#0;
   STAT36[102] := W#16#0;
   STAT36[103] := W#16#0;
   STAT36[104] := W#16#0;
   STAT36[105] := W#16#0;
   STAT36[106] := W#16#0;
   STAT36[107] := W#16#0;
   STAT36[108] := W#16#0;
   STAT36[109] := W#16#0;
   STAT36[110] := W#16#0;
   STAT36[111] := W#16#0;
   STAT36[112] := W#16#0;
   STAT36[113] := W#16#0;
   STAT36[114] := W#16#0;
   STAT36[115] := W#16#0;
   STAT36[116] := W#16#0;
   STAT36[117] := W#16#0;
   STAT36[118] := W#16#0;
   STAT36[119] := W#16#0;
   STAT36[120] := W#16#0;
   STAT36[121] := W#16#0;
   STAT36[122] := W#16#0;
   STAT36[123] := W#16#0;
   STAT36[124] := W#16#0;
   STAT36[125] := W#16#0;
   STAT36[126] := W#16#0;
   STAT36[127] := W#16#0;
   STAT36[128] := W#16#0;
   STAT36[129] := W#16#0;
   STAT36[130] := W#16#0;
   STAT36[131] := W#16#0;
   STAT36[132] := W#16#0;
   STAT36[133] := W#16#0;
   STAT36[134] := W#16#0;
   STAT36[135] := W#16#0;
   STAT36[136] := W#16#0;
   STAT36[137] := W#16#0;
   STAT36[138] := W#16#0;
   STAT36[139] := W#16#0;
   STAT36[140] := W#16#0;
   STAT36[141] := W#16#0;
   STAT36[142] := W#16#0;
   STAT36[143] := W#16#0;
   STAT36[144] := W#16#0;
   STAT36[145] := W#16#0;
   STAT36[146] := W#16#0;
   STAT36[147] := W#16#0;
   STAT36[148] := W#16#0;
   STAT36[149] := W#16#0;
   STAT36[150] := W#16#0;
   STAT36[151] := W#16#0;
   STAT36[152] := W#16#0;
   STAT36[153] := W#16#0;
   STAT36[154] := W#16#0;
   STAT36[155] := W#16#0;
   STAT36[156] := W#16#0;
   STAT36[157] := W#16#0;
   STAT36[158] := W#16#0;
   STAT36[159] := W#16#0;
   STAT36[160] := W#16#0;
   STAT36[161] := W#16#0;
   STAT36[162] := W#16#0;
   STAT36[163] := W#16#0;
   STAT36[164] := W#16#0;
   STAT36[165] := W#16#0;
   STAT36[166] := W#16#0;
   STAT36[167] := W#16#0;
   STAT36[168] := W#16#0;
   STAT36[169] := W#16#0;
   STAT36[170] := W#16#0;
   STAT36[171] := W#16#0;
   STAT36[172] := W#16#0;
   STAT36[173] := W#16#0;
   STAT36[174] := W#16#0;
   STAT36[175] := W#16#0;
   STAT36[176] := W#16#0;
   STAT36[177] := W#16#0;
   STAT36[178] := W#16#0;
   STAT36[179] := W#16#0;
   STAT36[180] := W#16#0;
   STAT36[181] := W#16#0;
   STAT36[182] := W#16#0;
   STAT36[183] := W#16#0;
   STAT36[184] := W#16#0;
   STAT36[185] := W#16#0;
   STAT36[186] := W#16#0;
   STAT36[187] := W#16#0;
   STAT36[188] := W#16#0;
   STAT36[189] := W#16#0;
   STAT36[190] := W#16#0;
   STAT36[191] := W#16#0;
   STAT36[192] := W#16#0;
   STAT36[193] := W#16#0;
   STAT36[194] := W#16#0;
   STAT36[195] := W#16#0;
   STAT36[196] := W#16#0;
   STAT36[197] := W#16#0;
   STAT36[198] := W#16#0;
   STAT36[199] := W#16#0;
   STAT36[200] := W#16#0;
   STAT36[201] := W#16#0;
   STAT36[202] := W#16#0;
   STAT36[203] := W#16#0;
   STAT36[204] := W#16#0;
   STAT36[205] := W#16#0;
   STAT36[206] := W#16#0;
   STAT36[207] := W#16#0;
   STAT36[208] := W#16#0;
   STAT36[209] := W#16#0;
   STAT36[210] := W#16#0;
   STAT36[211] := W#16#0;
   STAT36[212] := W#16#0;
   STAT36[213] := W#16#0;
   STAT36[214] := W#16#0;
   STAT36[215] := W#16#0;
   STAT36[216] := W#16#0;
   STAT36[217] := W#16#0;
   STAT36[218] := W#16#0;
   STAT36[219] := W#16#0;
   STAT36[220] := W#16#0;
   STAT36[221] := W#16#0;
   STAT36[222] := W#16#0;
   STAT36[223] := W#16#0;
   STAT36[224] := W#16#0;
   STAT36[225] := W#16#0;
   STAT36[226] := W#16#0;
   STAT36[227] := W#16#0;
   STAT36[228] := W#16#0;
   STAT36[229] := W#16#0;
   STAT36[230] := W#16#0;
   STAT36[231] := W#16#0;
   STAT36[232] := W#16#0;
   STAT36[233] := W#16#0;
   STAT36[234] := W#16#0;
   STAT36[235] := W#16#0;
   STAT36[236] := W#16#0;
   STAT36[237] := W#16#0;
   STAT36[238] := W#16#0;
   STAT36[239] := W#16#0;
   STAT36[240] := W#16#0;
   STAT36[241] := W#16#0;
   STAT36[242] := W#16#0;
   STAT36[243] := W#16#0;
   STAT36[244] := W#16#0;
   STAT36[245] := W#16#0;
   STAT36[246] := W#16#0;
   STAT36[247] := W#16#0;
   STAT36[248] := W#16#0;
   STAT36[249] := W#16#0;
   STAT36[250] := W#16#0;
   STAT36[251] := W#16#0;
   STAT36[252] := W#16#0;
   STAT36[253] := W#16#0;
   STAT36[254] := W#16#0;
   STAT36[255] := W#16#0;
   STAT36[256] := W#16#0;
   STAT36[257] := W#16#0;
   STAT36[258] := W#16#0;
   STAT36[259] := W#16#0;
   STAT36[260] := W#16#0;
   STAT36[261] := W#16#0;
   STAT36[262] := W#16#0;
   STAT36[263] := W#16#0;
   STAT36[264] := W#16#0;
   STAT36[265] := W#16#0;
   STAT36[266] := W#16#0;
   STAT36[267] := W#16#0;
   STAT36[268] := W#16#0;
   STAT36[269] := W#16#0;
   STAT36[270] := W#16#0;
   STAT36[271] := W#16#0;
   STAT36[272] := W#16#0;
   STAT36[273] := W#16#0;
   STAT36[274] := W#16#0;
   STAT36[275] := W#16#0;
   STAT36[276] := W#16#0;
   STAT36[277] := W#16#0;
   STAT36[278] := W#16#0;
   STAT36[279] := W#16#0;
   STAT36[280] := W#16#0;
   STAT36[281] := W#16#0;
   STAT36[282] := W#16#0;
   STAT36[283] := W#16#0;
   STAT36[284] := W#16#0;
   STAT36[285] := W#16#0;
   STAT36[286] := W#16#0;
   STAT36[287] := W#16#0;
   STAT36[288] := W#16#0;
   STAT36[289] := W#16#0;
   STAT36[290] := W#16#0;
   STAT36[291] := W#16#0;
   STAT36[292] := W#16#0;
   STAT36[293] := W#16#0;
   STAT36[294] := W#16#0;
   STAT36[295] := W#16#0;
   STAT36[296] := W#16#0;
   STAT36[297] := W#16#0;
   STAT36[298] := W#16#0;
   STAT36[299] := W#16#0;
   STAT36[300] := W#16#0;
   STAT36[301] := W#16#0;
   STAT36[302] := W#16#0;
   STAT36[303] := W#16#0;
   STAT36[304] := W#16#0;
   STAT36[305] := W#16#0;
   STAT36[306] := W#16#0;
   STAT36[307] := W#16#0;
   STAT36[308] := W#16#0;
   STAT36[309] := W#16#0;
   STAT36[310] := W#16#0;
   STAT36[311] := W#16#0;
   STAT36[312] := W#16#0;
   STAT36[313] := W#16#0;
   STAT36[314] := W#16#0;
   STAT36[315] := W#16#0;
   STAT36[316] := W#16#0;
   STAT36[317] := W#16#0;
   STAT36[318] := W#16#0;
   STAT36[319] := W#16#0;
   STAT36[320] := W#16#0;
   STAT36[321] := W#16#0;
   STAT36[322] := W#16#0;
   STAT36[323] := W#16#0;
   STAT36[324] := W#16#0;
   STAT36[325] := W#16#0;
   STAT36[326] := W#16#0;
   STAT36[327] := W#16#0;
   STAT36[328] := W#16#0;
   STAT36[329] := W#16#0;
   STAT36[330] := W#16#0;
   STAT36[331] := W#16#0;
   STAT36[332] := W#16#0;
   STAT36[333] := W#16#0;
   STAT36[334] := W#16#0;
   STAT36[335] := W#16#0;
   STAT36[336] := W#16#0;
   STAT36[337] := W#16#0;
   STAT36[338] := W#16#0;
   STAT36[339] := W#16#0;
   STAT36[340] := W#16#0;
   STAT36[341] := W#16#0;
   STAT36[342] := W#16#0;
   STAT36[343] := W#16#0;
   STAT36[344] := W#16#0;
   STAT36[345] := W#16#0;
   STAT36[346] := W#16#0;
   STAT36[347] := W#16#0;
   STAT36[348] := W#16#0;
   STAT36[349] := W#16#0;
   STAT36[350] := W#16#0;
   STAT36[351] := W#16#0;
   STAT36[352] := W#16#0;
   STAT36[353] := W#16#0;
   STAT36[354] := W#16#0;
   STAT36[355] := W#16#0;
   STAT36[356] := W#16#0;
   STAT36[357] := W#16#0;
   STAT36[358] := W#16#0;
   STAT36[359] := W#16#0;
   STAT36[360] := W#16#0;
   STAT36[361] := W#16#0;
   STAT36[362] := W#16#0;
   STAT36[363] := W#16#0;
   STAT36[364] := W#16#0;
   STAT36[365] := W#16#0;
   STAT36[366] := W#16#0;
   STAT36[367] := W#16#0;
   STAT36[368] := W#16#0;
   STAT36[369] := W#16#0;
   STAT36[370] := W#16#0;
   STAT36[371] := W#16#0;
   STAT36[372] := W#16#0;
   STAT36[373] := W#16#0;
   STAT36[374] := W#16#0;
   STAT36[375] := W#16#0;
   STAT36[376] := W#16#0;
   STAT36[377] := W#16#0;
   STAT36[378] := W#16#0;
   STAT36[379] := W#16#0;
   STAT36[380] := W#16#0;
   STAT36[381] := W#16#0;
   STAT36[382] := W#16#0;
   STAT36[383] := W#16#0;
   STAT36[384] := W#16#0;
   STAT36[385] := W#16#0;
   STAT36[386] := W#16#0;
   STAT36[387] := W#16#0;
   STAT36[388] := W#16#0;
   STAT36[389] := W#16#0;
   STAT36[390] := W#16#0;
   STAT36[391] := W#16#0;
   STAT36[392] := W#16#0;
   STAT36[393] := W#16#0;
   STAT36[394] := W#16#0;
   STAT36[395] := W#16#0;
   STAT36[396] := W#16#0;
   STAT36[397] := W#16#0;
   STAT36[398] := W#16#0;
   STAT36[399] := W#16#0;
   STAT36[400] := W#16#0;
   STAT36[401] := W#16#0;
   STAT36[402] := W#16#0;
   STAT36[403] := W#16#0;
   STAT36[404] := W#16#0;
   STAT36[405] := W#16#0;
   STAT36[406] := W#16#0;
   STAT36[407] := W#16#0;
   STAT36[408] := W#16#0;
   STAT36[409] := W#16#0;
   STAT36[410] := W#16#0;
   STAT36[411] := W#16#0;
   STAT36[412] := W#16#0;
   STAT36[413] := W#16#0;
   STAT36[414] := W#16#0;
   STAT36[415] := W#16#0;
   STAT36[416] := W#16#0;
   STAT36[417] := W#16#0;
   STAT36[418] := W#16#0;
   STAT36[419] := W#16#0;
   STAT36[420] := W#16#0;
   STAT36[421] := W#16#0;
   STAT36[422] := W#16#0;
   STAT36[423] := W#16#0;
   STAT36[424] := W#16#0;
   STAT36[425] := W#16#0;
   STAT36[426] := W#16#0;
   STAT36[427] := W#16#0;
   STAT36[428] := W#16#0;
   STAT36[429] := W#16#0;
   STAT36[430] := W#16#0;
   STAT36[431] := W#16#0;
   STAT36[432] := W#16#0;
   STAT36[433] := W#16#0;
   STAT36[434] := W#16#0;
   STAT36[435] := W#16#0;
   STAT36[436] := W#16#0;
   STAT36[437] := W#16#0;
   STAT36[438] := W#16#0;
   STAT36[439] := W#16#0;
   STAT36[440] := W#16#0;
   STAT36[441] := W#16#0;
   STAT36[442] := W#16#0;
   STAT36[443] := W#16#0;
   STAT36[444] := W#16#0;
   STAT36[445] := W#16#0;
   STAT36[446] := W#16#0;
   STAT36[447] := W#16#0;
   STAT36[448] := W#16#0;
   STAT36[449] := W#16#0;
   STAT36[450] := W#16#0;
   STAT36[451] := W#16#0;
   STAT36[452] := W#16#0;
   STAT36[453] := W#16#0;
   STAT36[454] := W#16#0;
   STAT36[455] := W#16#0;
   STAT36[456] := W#16#0;
   STAT36[457] := W#16#0;
   STAT36[458] := W#16#0;
   STAT36[459] := W#16#0;
   STAT36[460] := W#16#0;
   STAT36[461] := W#16#0;
   STAT36[462] := W#16#0;
   STAT36[463] := W#16#0;
   STAT36[464] := W#16#0;
   STAT36[465] := W#16#0;
   STAT36[466] := W#16#0;
   STAT36[467] := W#16#0;
   STAT36[468] := W#16#0;
   STAT36[469] := W#16#0;
   STAT36[470] := W#16#0;
   STAT36[471] := W#16#0;
   STAT36[472] := W#16#0;
   STAT36[473] := W#16#0;
   STAT36[474] := W#16#0;
   STAT36[475] := W#16#0;
   STAT36[476] := W#16#0;
   STAT36[477] := W#16#0;
   STAT36[478] := W#16#0;
   STAT36[479] := W#16#0;
   STAT36[480] := W#16#0;
   STAT36[481] := W#16#0;
   STAT36[482] := W#16#0;
   STAT36[483] := W#16#0;
   STAT36[484] := W#16#0;
   STAT36[485] := W#16#0;
   STAT36[486] := W#16#0;
   STAT36[487] := W#16#0;
   STAT36[488] := W#16#0;
   STAT36[489] := W#16#0;
   STAT36[490] := W#16#0;
   STAT36[491] := W#16#0;
   STAT36[492] := W#16#0;
   STAT36[493] := W#16#0;
   STAT36[494] := W#16#0;
   STAT36[495] := W#16#0;
   STAT36[496] := W#16#0;
   STAT36[497] := W#16#0;
   STAT36[498] := W#16#0;
   STAT36[499] := W#16#0;
   STAT36[500] := W#16#0;
   STAT37[1] := B#16#0;
   STAT37[2] := B#16#0;
   STAT37[3] := B#16#0;
   STAT37[4] := B#16#0;
   STAT37[5] := B#16#0;
   STAT37[6] := B#16#0;
   STAT37[7] := B#16#0;
   STAT37[8] := B#16#0;
   STAT37[9] := B#16#0;
   STAT37[10] := B#16#0;
   STAT37[11] := B#16#0;
   STAT37[12] := B#16#0;
   STAT37[13] := B#16#0;
   STAT37[14] := B#16#0;
   STAT37[15] := B#16#0;
   STAT37[16] := B#16#0;
   STAT38[1] := B#16#0;
   STAT38[2] := B#16#0;
   STAT38[3] := B#16#0;
   STAT38[4] := B#16#0;
   STAT39[1] := B#16#0;
   STAT39[2] := B#16#0;
   STAT39[3] := B#16#0;
   STAT39[4] := B#16#0;
   STAT39[5] := B#16#0;
   STAT39[6] := B#16#0;
   STAT39[7] := B#16#0;
   STAT39[8] := B#16#0;
   STAT39[9] := B#16#0;
   STAT39[10] := B#16#0;
   STAT39[11] := B#16#0;
   STAT39[12] := B#16#0;
   STAT39[13] := B#16#0;
   STAT39[14] := B#16#0;
   STAT39[15] := B#16#0;
   STAT39[16] := B#16#0;
END_DATA_BLOCK

DATA_BLOCK DB 253
TITLE =
VERSION : 0.1


  STRUCT
   DB_VAR : ARRAY  [0 .. 99 ] OF WORD ;
  END_STRUCT ;
BEGIN
   DB_VAR[0] := W#16#0;
   DB_VAR[1] := W#16#0;
   DB_VAR[2] := W#16#0;
   DB_VAR[3] := W#16#87;
   DB_VAR[4] := W#16#2718;
   DB_VAR[5] := W#16#2222;
   DB_VAR[6] := W#16#87;
   DB_VAR[7] := W#16#2717;
   DB_VAR[8] := W#16#220A;
   DB_VAR[9] := W#16#87;
   DB_VAR[10] := W#16#2716;
   DB_VAR[11] := W#16#2222;
   DB_VAR[12] := W#16#0;
   DB_VAR[13] := W#16#0;
   DB_VAR[14] := W#16#0;
   DB_VAR[15] := W#16#87;
   DB_VAR[16] := W#16#2715;
   DB_VAR[17] := W#16#2222;
   DB_VAR[18] := W#16#87;
   DB_VAR[19] := W#16#2714;
   DB_VAR[20] := W#16#2222;
   DB_VAR[21] := W#16#87;
   DB_VAR[22] := W#16#2713;
   DB_VAR[23] := W#16#220A;
   DB_VAR[24] := W#16#87;
   DB_VAR[25] := W#16#2712;
   DB_VAR[26] := W#16#2222;
   DB_VAR[27] := W#16#87;
   DB_VAR[28] := W#16#2711;
   DB_VAR[29] := W#16#2284;
   DB_VAR[30] := W#16#87;
   DB_VAR[31] := W#16#2710;
   DB_VAR[32] := W#16#2222;
   DB_VAR[33] := W#16#87;
   DB_VAR[34] := W#16#2709;
   DB_VAR[35] := W#16#220A;
   DB_VAR[36] := W#16#0;
   DB_VAR[37] := W#16#0;
   DB_VAR[38] := W#16#0;
   DB_VAR[39] := W#16#87;
   DB_VAR[40] := W#16#2708;
   DB_VAR[41] := W#16#2222;
   DB_VAR[42] := W#16#0;
   DB_VAR[43] := W#16#0;
   DB_VAR[44] := W#16#0;
   DB_VAR[45] := W#16#0;
   DB_VAR[46] := W#16#0;
   DB_VAR[47] := W#16#0;
   DB_VAR[48] := W#16#0;
   DB_VAR[49] := W#16#0;
   DB_VAR[50] := W#16#0;
   DB_VAR[51] := W#16#0;
   DB_VAR[52] := W#16#0;
   DB_VAR[53] := W#16#0;
   DB_VAR[54] := W#16#0;
   DB_VAR[55] := W#16#0;
   DB_VAR[56] := W#16#0;
   DB_VAR[57] := W#16#0;
   DB_VAR[58] := W#16#0;
   DB_VAR[59] := W#16#0;
   DB_VAR[60] := W#16#0;
   DB_VAR[61] := W#16#0;
   DB_VAR[62] := W#16#0;
   DB_VAR[63] := W#16#0;
   DB_VAR[64] := W#16#0;
   DB_VAR[65] := W#16#0;
   DB_VAR[66] := W#16#0;
   DB_VAR[67] := W#16#0;
   DB_VAR[68] := W#16#0;
   DB_VAR[69] := W#16#0;
   DB_VAR[70] := W#16#0;
   DB_VAR[71] := W#16#0;
   DB_VAR[72] := W#16#0;
   DB_VAR[73] := W#16#0;
   DB_VAR[74] := W#16#0;
   DB_VAR[75] := W#16#0;
   DB_VAR[76] := W#16#0;
   DB_VAR[77] := W#16#0;
   DB_VAR[78] := W#16#0;
   DB_VAR[79] := W#16#0;
   DB_VAR[80] := W#16#0;
   DB_VAR[81] := W#16#0;
   DB_VAR[82] := W#16#0;
   DB_VAR[83] := W#16#0;
   DB_VAR[84] := W#16#0;
   DB_VAR[85] := W#16#0;
   DB_VAR[86] := W#16#0;
   DB_VAR[87] := W#16#0;
   DB_VAR[88] := W#16#0;
   DB_VAR[89] := W#16#0;
   DB_VAR[90] := W#16#0;
   DB_VAR[91] := W#16#0;
   DB_VAR[92] := W#16#0;
   DB_VAR[93] := W#16#0;
   DB_VAR[94] := W#16#0;
   DB_VAR[95] := W#16#0;
   DB_VAR[96] := W#16#0;
   DB_VAR[97] := W#16#0;
   DB_VAR[98] := W#16#0;
   DB_VAR[99] := W#16#0;
END_DATA_BLOCK

DATA_BLOCK DB 261
VERSION : 0.1


